LIN {X 0,Y 567.245,Z 796.089,A -85,B 0,C 180,E1 -2627.298,E2 -2627.298} C_VEL
LIN {X 0,Y 567.525,Z 782.898,A -85,B 0,C 180,E1 -2628.314,E2 -2628.314} C_VEL
LIN {X 0,Y 567.877,Z 768.842,A -85,B 0,C 180,E1 -2629.238,E2 -2629.238} C_VEL
LIN {X 0,Y 568.254,Z 752.432,A -85,B 0,C 180,E1 -2630.132,E2 -2630.132} C_VEL
LIN {X 0,Y 568.541,Z 736.853,A -85,B 0,C 180,E1 -2630.817,E2 -2630.817} C_VEL
LIN {X 0,Y 568.789,Z 721.335,A -85,B 0,C 180,E1 -2631.353,E2 -2631.353} C_VEL
LIN {X 0,Y 569.036,Z 705.143,A -85,B 0,C 180,E1 -2631.778,E2 -2631.778} C_VEL
LIN {X 0,Y 569.217,Z 685.553,A -85,B 0,C 180,E1 -2632.108,E2 -2632.108} C_VEL
LIN {X 0,Y 569.98,Z 494.969,A -85,B 0,C 180,E1 -2634.639,E2 -2634.639} C_VEL
LIN {X 0,Y 569.683,Z 492.167,A -85,B 0,C 180,E1 -2634.691,E2 -2634.691} C_VEL
LIN {X 0,Y 567.818,Z 484.792,A -85,B 0,C 180,E1 -2634.886,E2 -2634.886} C_VEL
LIN {X 0,Y 567.716,Z 483.349,A -85,B 0,C 180,E1 -2635.005,E2 -2635.005} C_VEL
LIN {X 0,Y 568.103,Z 461.779,A -85,B 0,C 180,E1 -2637.839,E2 -2637.839} C_VEL
LIN {X 0,Y 568.437,Z 446.604,A -85,B 0,C 180,E1 -2639.873,E2 -2639.873} C_VEL
LIN {X 0,Y 566.233,Z 437.352,A -85,B 0,C 180,E1 -2641.317,E2 -2641.317} C_VEL
LIN {X 0,Y 566.208,Z 437.196,A -85,B 0,C 180,E1 -2643.955,E2 -2643.955} C_VEL
LIN {X 0,Y 566.212,Z 437.2,A -85,B 0,C 180,E1 -2646.568,E2 -2646.568} C_VEL
LIN {X 0,Y 566.207,Z 437.206,A -85,B 0,C 180,E1 -2649.685,E2 -2649.685} C_VEL
LIN {X 0,Y 566.185,Z 437.205,A -85,B 0,C 180,E1 -2652.089,E2 -2652.089} C_VEL
LIN {X 0,Y 566.167,Z 437.206,A -85,B 0,C 180,E1 -2655.035,E2 -2655.035} C_VEL
LIN {X 0,Y 566.208,Z 437.208,A -85,B 0,C 180,E1 -2657.912,E2 -2657.912} C_VEL
LIN {X 0,Y 566.217,Z 437.197,A -85,B 0,C 180,E1 -2660.727,E2 -2660.727} C_VEL
LIN {X 0,Y 566.211,Z 437.207,A -85,B 0,C 180,E1 -2663.783,E2 -2663.783} C_VEL
LIN {X 0,Y 566.204,Z 437.204,A -85,B 0,C 180,E1 -2666.265,E2 -2666.265} C_VEL
LIN {X 0,Y 566.195,Z 437.201,A -85,B 0,C 180,E1 -2668.921,E2 -2668.921} C_VEL
LIN {X 0,Y 566.186,Z 437.196,A -85,B 0,C 180,E1 -2671.046,E2 -2671.046} C_VEL
LIN {X 0,Y 566.236,Z 437.194,A -85,B 0,C 180,E1 -2673.46,E2 -2673.46} C_VEL
LIN {X 0,Y 566.191,Z 437.208,A -85,B 0,C 180,E1 -2675.819,E2 -2675.819} C_VEL
LIN {X 0,Y 566.208,Z 437.192,A -85,B 0,C 180,E1 -2678.902,E2 -2678.902} C_VEL
LIN {X 0,Y 566.204,Z 437.194,A -85,B 0,C 180,E1 -2681.172,E2 -2681.172} C_VEL
LIN {X 0,Y 566.211,Z 437.199,A -85,B 0,C 180,E1 -2683.412,E2 -2683.412} C_VEL
LIN {X 0,Y 566.19,Z 437.208,A -85,B 0,C 180,E1 -2686.359,E2 -2686.359} C_VEL
LIN {X 0,Y 566.266,Z 437.197,A -85,B 0,C 180,E1 -2688.654,E2 -2688.654} C_VEL
LIN {X 0,Y 566.24,Z 437.193,A -85,B 0,C 180,E1 -2691.434,E2 -2691.434} C_VEL
LIN {X 0,Y 566.25,Z 437.203,A -85,B 0,C 180,E1 -2694.302,E2 -2694.302} C_VEL
LIN {X 0,Y 566.271,Z 437.192,A -85,B 0,C 180,E1 -2697.866,E2 -2697.866} C_VEL
LIN {X 0,Y 566.298,Z 437.192,A -85,B 0,C 180,E1 -2700.711,E2 -2700.711} C_VEL
LIN {X 0,Y 566.27,Z 437.197,A -85,B 0,C 180,E1 -2702.845,E2 -2702.845} C_VEL
LIN {X 0,Y 566.258,Z 437.191,A -85,B 0,C 180,E1 -2705.698,E2 -2705.698} C_VEL
LIN {X 0,Y 566.24,Z 437.204,A -85,B 0,C 180,E1 -2708.565,E2 -2708.565} C_VEL
LIN {X 0,Y 566.241,Z 437.194,A -85,B 0,C 180,E1 -2711.454,E2 -2711.454} C_VEL
LIN {X 0,Y 566.223,Z 437.204,A -85,B 0,C 180,E1 -2714.507,E2 -2714.507} C_VEL
LIN {X 0,Y 566.194,Z 437.204,A -85,B 0,C 180,E1 -2717.332,E2 -2717.332} C_VEL
LIN {X 0,Y 566.21,Z 437.201,A -85,B 0,C 180,E1 -2720.337,E2 -2720.337} C_VEL
LIN {X 0,Y 566.18,Z 437.205,A -85,B 0,C 180,E1 -2723.404,E2 -2723.404} C_VEL
LIN {X 0,Y 566.215,Z 437.192,A -85,B 0,C 180,E1 -2725.749,E2 -2725.749} C_VEL
LIN {X 0,Y 566.208,Z 437.198,A -85,B 0,C 180,E1 -2727.495,E2 -2727.495} C_VEL
LIN {X 0,Y 565.53,Z 437.283,A -85,B 0,C 180,E1 -2728.089,E2 -2728.089} C_VEL
LIN {X 0,Y 562.664,Z 437.649,A -85,B 0,C 180,E1 -2729.052,E2 -2729.052} C_VEL
LIN {X 0,Y 560.253,Z 437.945,A -85,B 0,C 180,E1 -2729.828,E2 -2729.828} C_VEL
LIN {X 0,Y 559.224,Z 438.072,A -85,B 0,C 180,E1 -2730.427,E2 -2730.427} C_VEL
LIN {X 0,Y 559.144,Z 438.083,A -85,B 0,C 180,E1 -2730.629,E2 -2730.629} C_VEL
LIN {X 0,Y 559.155,Z 438.071,A -85,B 0,C 180,E1 -2733.575,E2 -2733.575} C_VEL
LIN {X 0,Y 559.16,Z 438.078,A -85,B 0,C 180,E1 -2736.449,E2 -2736.449} C_VEL
LIN {X 0,Y 559.171,Z 438.084,A -85,B 0,C 180,E1 -2738.934,E2 -2738.934} C_VEL
LIN {X 0,Y 559.189,Z 438.077,A -85,B 0,C 180,E1 -2741.767,E2 -2741.767} C_VEL
LIN {X 0,Y 559.132,Z 438.085,A -85,B 0,C 180,E1 -2744.739,E2 -2744.739} C_VEL
LIN {X 0,Y 559.169,Z 438.079,A -85,B 0,C 180,E1 -2747.863,E2 -2747.863} C_VEL
LIN {X 0,Y 559.178,Z 438.076,A -85,B 0,C 180,E1 -2750.135,E2 -2750.135} C_VEL
LIN {X 0,Y 559.14,Z 438.084,A -85,B 0,C 180,E1 -2752.893,E2 -2752.893} C_VEL
LIN {X 0,Y 559.156,Z 438.087,A -85,B 0,C 180,E1 -2755.557,E2 -2755.557} C_VEL
LIN {X 0,Y 559.165,Z 438.079,A -85,B 0,C 180,E1 -2758.138,E2 -2758.138} C_VEL
LIN {X 0,Y 559.138,Z 438.081,A -85,B 0,C 180,E1 -2760.647,E2 -2760.647} C_VEL
LIN {X 0,Y 559.177,Z 438.081,A -85,B 0,C 180,E1 -2763.17,E2 -2763.17} C_VEL
LIN {X 0,Y 559.152,Z 438.088,A -85,B 0,C 180,E1 -2765.495,E2 -2765.495} C_VEL
LIN {X 0,Y 559.167,Z 438.077,A -85,B 0,C 180,E1 -2768.624,E2 -2768.624} C_VEL
LIN {X 0,Y 559.167,Z 438.079,A -85,B 0,C 180,E1 -2770.927,E2 -2770.927} C_VEL
LIN {X 0,Y 559.166,Z 438.085,A -85,B 0,C 180,E1 -2773.948,E2 -2773.948} C_VEL
LIN {X 0,Y 559.171,Z 438.081,A -85,B 0,C 180,E1 -2776.184,E2 -2776.184} C_VEL
LIN {X 0,Y 559.19,Z 438.076,A -85,B 0,C 180,E1 -2779.134,E2 -2779.134} C_VEL
LIN {X 0,Y 559.202,Z 438.081,A -85,B 0,C 180,E1 -2782.054,E2 -2782.054} C_VEL
LIN {X 0,Y 559.249,Z 438.068,A -85,B 0,C 180,E1 -2784.953,E2 -2784.953} C_VEL
LIN {X 0,Y 559.251,Z 438.076,A -85,B 0,C 180,E1 -2787.839,E2 -2787.839} C_VEL
LIN {X 0,Y 559.267,Z 438.066,A -85,B 0,C 180,E1 -2790.72,E2 -2790.72} C_VEL
LIN {X 0,Y 559.235,Z 438.07,A -85,B 0,C 180,E1 -2792.881,E2 -2792.881} C_VEL
LIN {X 0,Y 559.225,Z 438.076,A -85,B 0,C 180,E1 -2795.77,E2 -2795.77} C_VEL
LIN {X 0,Y 559.184,Z 438.078,A -85,B 0,C 180,E1 -2798.674,E2 -2798.674} C_VEL
LIN {X 0,Y 559.202,Z 438.076,A -85,B 0,C 180,E1 -2801.6,E2 -2801.6} C_VEL
LIN {X 0,Y 559.196,Z 438.079,A -85,B 0,C 180,E1 -2804.595,E2 -2804.595} C_VEL
LIN {X 0,Y 559.159,Z 438.079,A -85,B 0,C 180,E1 -2807.556,E2 -2807.556} C_VEL
LIN {X 0,Y 559.168,Z 438.081,A -85,B 0,C 180,E1 -2809.837,E2 -2809.837} C_VEL
LIN {X 0,Y 559.137,Z 438.088,A -85,B 0,C 180,E1 -2812.152,E2 -2812.152} C_VEL
LIN {X 0,Y 559.173,Z 438.077,A -85,B 0,C 180,E1 -2815.298,E2 -2815.298} C_VEL
LIN {X 0,Y 559.19,Z 438.076,A -85,B 0,C 180,E1 -2817.711,E2 -2817.711} C_VEL
LIN {X 0,Y 559.156,Z 438.082,A -85,B 0,C 180,E1 -2821.018,E2 -2821.018} C_VEL
LIN {X 0,Y 559.172,Z 438.079,A -85,B 0,C 180,E1 -2823.951,E2 -2823.951} C_VEL
LIN {X 0,Y 559.162,Z 438.085,A -85,B 0,C 180,E1 -2826.448,E2 -2826.448} C_VEL
LIN {X 0,Y 559.171,Z 438.083,A -85,B 0,C 180,E1 -2828.933,E2 -2828.933} C_VEL
LIN {X 0,Y 559.184,Z 438.075,A -85,B 0,C 180,E1 -2831.767,E2 -2831.767} C_VEL
LIN {X 0,Y 559.132,Z 438.091,A -85,B 0,C 180,E1 -2834.739,E2 -2834.739} C_VEL
LIN {X 0,Y 559.156,Z 438.082,A -85,B 0,C 180,E1 -2837.257,E2 -2837.257} C_VEL
LIN {X 0,Y 559.178,Z 438.077,A -85,B 0,C 180,E1 -2840.135,E2 -2840.135} C_VEL
LIN {X 0,Y 559.139,Z 438.09,A -85,B 0,C 180,E1 -2842.892,E2 -2842.892} C_VEL
LIN {X 0,Y 559.147,Z 438.071,A -85,B 0,C 180,E1 -2845.556,E2 -2845.556} C_VEL
LIN {X 0,Y 559.162,Z 438.076,A -85,B 0,C 180,E1 -2848.137,E2 -2848.137} C_VEL
LIN {X 0,Y 559.149,Z 438.084,A -85,B 0,C 180,E1 -2850.647,E2 -2850.647} C_VEL
LIN {X 0,Y 559.173,Z 438.074,A -85,B 0,C 180,E1 -2853.17,E2 -2853.17} C_VEL
LIN {X 0,Y 559.148,Z 438.082,A -85,B 0,C 180,E1 -2855.495,E2 -2855.495} C_VEL
LIN {X 0,Y 559.167,Z 438.079,A -85,B 0,C 180,E1 -2858.624,E2 -2858.624} C_VEL
LIN {X 0,Y 559.162,Z 438.082,A -85,B 0,C 180,E1 -2860.926,E2 -2860.926} C_VEL
LIN {X 0,Y 559.16,Z 438.075,A -85,B 0,C 180,E1 -2863.948,E2 -2863.948} C_VEL
LIN {X 0,Y 559.163,Z 438.077,A -85,B 0,C 180,E1 -2866.184,E2 -2866.184} C_VEL
LIN {X 0,Y 559.202,Z 438.077,A -85,B 0,C 180,E1 -2869.134,E2 -2869.134} C_VEL
LIN {X 0,Y 559.2,Z 438.073,A -85,B 0,C 180,E1 -2872.054,E2 -2872.054} C_VEL
LIN {X 0,Y 559.253,Z 438.067,A -85,B 0,C 180,E1 -2874.954,E2 -2874.954} C_VEL
LIN {X 0,Y 559.242,Z 438.068,A -85,B 0,C 180,E1 -2877.84,E2 -2877.84} C_VEL
LIN {X 0,Y 559.267,Z 438.065,A -85,B 0,C 180,E1 -2880.72,E2 -2880.72} C_VEL
LIN {X 0,Y 559.236,Z 438.068,A -85,B 0,C 180,E1 -2882.882,E2 -2882.882} C_VEL
LIN {X 0,Y 559.22,Z 438.078,A -85,B 0,C 180,E1 -2885.77,E2 -2885.77} C_VEL
LIN {X 0,Y 559.195,Z 438.07,A -85,B 0,C 180,E1 -2888.674,E2 -2888.674} C_VEL
LIN {X 0,Y 559.2,Z 438.081,A -85,B 0,C 180,E1 -2891.601,E2 -2891.601} C_VEL
LIN {X 0,Y 559.19,Z 438.074,A -85,B 0,C 180,E1 -2894.596,E2 -2894.596} C_VEL
LIN {X 0,Y 559.155,Z 438.084,A -85,B 0,C 180,E1 -2897.557,E2 -2897.557} C_VEL
LIN {X 0,Y 559.166,Z 438.074,A -85,B 0,C 180,E1 -2899.838,E2 -2899.838} C_VEL
LIN {X 0,Y 559.133,Z 438.086,A -85,B 0,C 180,E1 -2902.153,E2 -2902.153} C_VEL
LIN {X 0,Y 559.171,Z 438.077,A -85,B 0,C 180,E1 -2905.188,E2 -2905.188} C_VEL
LIN {X 0,Y 559.186,Z 438.076,A -85,B 0,C 180,E1 -2907.712,E2 -2907.712} C_VEL
LIN {X 0,Y 559.16,Z 438.085,A -85,B 0,C 180,E1 -2910.182,E2 -2910.182} C_VEL
LIN {X 0,Y 559.167,Z 438.078,A -85,B 0,C 180,E1 -2912.714,E2 -2912.714} C_VEL
LIN {X 0,Y 559.149,Z 438.074,A -85,B 0,C 180,E1 -2915.322,E2 -2915.322} C_VEL
LIN {X 0,Y 559.129,Z 438.09,A -85,B 0,C 180,E1 -2918.018,E2 -2918.018} C_VEL
LIN {X 0,Y 559.17,Z 438.078,A -85,B 0,C 180,E1 -2920.811,E2 -2920.811} C_VEL
LIN {X 0,Y 559.156,Z 438.08,A -85,B 0,C 180,E1 -2923.732,E2 -2923.732} C_VEL
LIN {X 0,Y 559.14,Z 438.081,A -85,B 0,C 180,E1 -2926.804,E2 -2926.804} C_VEL
LIN {X 0,Y 559.171,Z 438.078,A -85,B 0,C 180,E1 -2929.19,E2 -2929.19} C_VEL
LIN {X 0,Y 559.129,Z 438.075,A -85,B 0,C 180,E1 -2931.983,E2 -2931.983} C_VEL
LIN {X 0,Y 559.155,Z 438.081,A -85,B 0,C 180,E1 -2934.784,E2 -2934.784} C_VEL
LIN {X 0,Y 559.171,Z 438.078,A -85,B 0,C 180,E1 -2937.362,E2 -2937.362} C_VEL
LIN {X 0,Y 559.189,Z 438.266,A -85,B 0,C 180,E1 -2938.379,E2 -2938.379} C_VEL
LIN {X 0,Y 561.701,Z 448.315,A -85,B 0,C 180,E1 -2939.969,E2 -2939.969} C_VEL
LIN {X 0,Y 561.228,Z 469.907,A -85,B 0,C 180,E1 -2942.89,E2 -2942.89} C_VEL
LIN {X 0,Y 560.941,Z 484.201,A -85,B 0,C 180,E1 -2944.76,E2 -2944.76} C_VEL
LIN {X 0,Y 563.361,Z 494.017,A -85,B 0,C 180,E1 -2945.038,E2 -2945.038} C_VEL
LIN {X 0,Y 563.124,Z 583.687,A -85,B 0,C 180,E1 -2946.257,E2 -2946.257} C_VEL
LIN {X 0,Y 562.553,Z 696.291,A -85,B 0,C 180,E1 -2947.784,E2 -2947.784} C_VEL
LIN {X 0,Y 562.302,Z 712.289,A -85,B 0,C 180,E1 -2948.124,E2 -2948.124} C_VEL
LIN {X 0,Y 562.001,Z 730.611,A -85,B 0,C 180,E1 -2948.689,E2 -2948.689} C_VEL
LIN {X 0,Y 561.681,Z 745.689,A -85,B 0,C 180,E1 -2949.3,E2 -2949.3} C_VEL
LIN {X 0,Y 561.376,Z 758.835,A -85,B 0,C 180,E1 -2949.952,E2 -2949.952} C_VEL
LIN {X 0,Y 560.948,Z 773.325,A -85,B 0,C 180,E1 -2950.8,E2 -2950.8} C_VEL
LIN {X 0,Y 560.595,Z 788.011,A -85,B 0,C 180,E1 -2951.83,E2 -2951.83} C_VEL
LIN {X 0,Y 560.163,Z 802.482,A -85,B 0,C 180,E1 -2953.043,E2 -2953.043} C_VEL
LIN {X 0,Y 559.862,Z 813.823,A -85,B 0,C 180,E1 -2954.156,E2 -2954.156} C_VEL
LIN {X 0,Y 559.584,Z 825.316,A -85,B 0,C 180,E1 -2955.453,E2 -2955.453} C_VEL
LIN {X 0,Y 559.326,Z 836.44,A -85,B 0,C 180,E1 -2956.929,E2 -2956.929} C_VEL
LIN {X 0,Y 559.15,Z 845.808,A -85,B 0,C 180,E1 -2958.399,E2 -2958.399} C_VEL
LIN {X 0,Y 559.013,Z 853.664,A -85,B 0,C 180,E1 -2959.863,E2 -2959.863} C_VEL
LIN {X 0,Y 558.908,Z 860.28,A -85,B 0,C 180,E1 -2961.321,E2 -2961.321} C_VEL
LIN {X 0,Y 558.889,Z 865.667,A -85,B 0,C 180,E1 -2962.776,E2 -2962.776} C_VEL
LIN {X 0,Y 558.863,Z 870.027,A -85,B 0,C 180,E1 -2964.226,E2 -2964.226} C_VEL
LIN {X 0,Y 558.803,Z 873.298,A -85,B 0,C 180,E1 -2965.672,E2 -2965.672} C_VEL
LIN {X 0,Y 558.79,Z 875.656,A -85,B 0,C 180,E1 -2967.116,E2 -2967.116} C_VEL
LIN {X 0,Y 558.738,Z 877.009,A -85,B 0,C 180,E1 -2968.559,E2 -2968.559} C_VEL
LIN {X 0,Y 558.734,Z 877.5,A -85,B 0,C 180,E1 -2970,E2 -2970} C_VEL
LIN {X 0,Y 558.738,Z 877.009,A -85,B 0,C 180,E1 -2971.441,E2 -2971.441} C_VEL
LIN {X 0,Y 558.79,Z 875.656,A -85,B 0,C 180,E1 -2972.884,E2 -2972.884} C_VEL
LIN {X 0,Y 558.802,Z 873.298,A -85,B 0,C 180,E1 -2974.328,E2 -2974.328} C_VEL
LIN {X 0,Y 558.863,Z 870.027,A -85,B 0,C 180,E1 -2975.774,E2 -2975.774} C_VEL
LIN {X 0,Y 558.889,Z 865.667,A -85,B 0,C 180,E1 -2977.224,E2 -2977.224} C_VEL
LIN {X 0,Y 558.908,Z 860.28,A -85,B 0,C 180,E1 -2978.679,E2 -2978.679} C_VEL
LIN {X 0,Y 559.013,Z 853.664,A -85,B 0,C 180,E1 -2980.137,E2 -2980.137} C_VEL
LIN {X 0,Y 559.162,Z 844.729,A -85,B 0,C 180,E1 -2981.785,E2 -2981.785} C_VEL
LIN {X 0,Y 559.359,Z 835.161,A -85,B 0,C 180,E1 -2983.256,E2 -2983.256} C_VEL
LIN {X 0,Y 559.59,Z 825.316,A -85,B 0,C 180,E1 -2984.547,E2 -2984.547} C_VEL
LIN {X 0,Y 559.861,Z 813.823,A -85,B 0,C 180,E1 -2985.844,E2 -2985.844} C_VEL
LIN {X 0,Y 560.199,Z 801.481,A -85,B 0,C 180,E1 -2987.049,E2 -2987.049} C_VEL
LIN {X 0,Y 560.622,Z 786.738,A -85,B 0,C 180,E1 -2988.264,E2 -2988.264} C_VEL
LIN {X 0,Y 560.948,Z 773.325,A -85,B 0,C 180,E1 -2989.2,E2 -2989.2} C_VEL
LIN {X 0,Y 561.341,Z 758.821,A -85,B 0,C 180,E1 -2990.05,E2 -2990.05} C_VEL
LIN {X 0,Y 561.711,Z 743.643,A -85,B 0,C 180,E1 -2990.794,E2 -2990.794} C_VEL
LIN {X 0,Y 562.108,Z 725.885,A -85,B 0,C 180,E1 -2991.475,E2 -2991.475} C_VEL
LIN {X 0,Y 562.367,Z 709.394,A -85,B 0,C 180,E1 -2991.946,E2 -2991.946} C_VEL
LIN {X 0,Y 562.577,Z 693.902,A -85,B 0,C 180,E1 -2992.256,E2 -2992.256} C_VEL
LIN {X 0,Y 563.53,Z 495.969,A -85,B 0,C 180,E1 -2994.927,E2 -2994.927} C_VEL
LIN {X 0,Y 563.082,Z 492.938,A -85,B 0,C 180,E1 -2994.99,E2 -2994.99} C_VEL
LIN {X 0,Y 560.987,Z 484.416,A -85,B 0,C 180,E1 -2995.225,E2 -2995.225} C_VEL
LIN {X 0,Y 561.064,Z 478.235,A -85,B 0,C 180,E1 -2996.002,E2 -2996.002} C_VEL
LIN {X 0,Y 561.525,Z 457.167,A -85,B 0,C 180,E1 -2998.823,E2 -2998.823} C_VEL
LIN {X 0,Y 561.698,Z 448.315,A -85,B 0,C 180,E1 -3000.031,E2 -3000.031} C_VEL
LIN {X 0,Y 559.214,Z 438.272,A -85,B 0,C 180,E1 -3001.619,E2 -3001.619} C_VEL
LIN {X 0,Y 559.153,Z 438.077,A -85,B 0,C 180,E1 -3004.443,E2 -3004.443} C_VEL
LIN {X 0,Y 559.142,Z 438.081,A -85,B 0,C 180,E1 -3007.107,E2 -3007.107} C_VEL
LIN {X 0,Y 559.164,Z 438.085,A -85,B 0,C 180,E1 -3009.942,E2 -3009.942} C_VEL
LIN {X 0,Y 559.152,Z 438.078,A -85,B 0,C 180,E1 -3012.743,E2 -3012.743} C_VEL
LIN {X 0,Y 559.149,Z 438.084,A -85,B 0,C 180,E1 -3015.76,E2 -3015.76} C_VEL
LIN {X 0,Y 559.186,Z 438.077,A -85,B 0,C 180,E1 -3018.232,E2 -3018.232} C_VEL
LIN {X 0,Y 559.172,Z 438.076,A -85,B 0,C 180,E1 -3021.19,E2 -3021.19} C_VEL
LIN {X 0,Y 559.165,Z 438.084,A -85,B 0,C 180,E1 -3023.791,E2 -3023.791} C_VEL
LIN {X 0,Y 559.157,Z 438.08,A -85,B 0,C 180,E1 -3026.425,E2 -3026.425} C_VEL
LIN {X 0,Y 559.158,Z 438.077,A -85,B 0,C 180,E1 -3028.981,E2 -3028.981} C_VEL
LIN {X 0,Y 559.162,Z 438.074,A -85,B 0,C 180,E1 -3031.618,E2 -3031.618} C_VEL
LIN {X 0,Y 559.19,Z 438.077,A -85,B 0,C 180,E1 -3033.903,E2 -3033.903} C_VEL
LIN {X 0,Y 559.148,Z 438.081,A -85,B 0,C 180,E1 -3036.567,E2 -3036.567} C_VEL
LIN {X 0,Y 559.177,Z 438.067,A -85,B 0,C 180,E1 -3039.395,E2 -3039.395} C_VEL
LIN {X 0,Y 559.146,Z 438.075,A -85,B 0,C 180,E1 -3041.686,E2 -3041.686} C_VEL
LIN {X 0,Y 559.161,Z 438.082,A -85,B 0,C 180,E1 -3043.948,E2 -3043.948} C_VEL
LIN {X 0,Y 559.164,Z 438.084,A -85,B 0,C 180,E1 -3046.184,E2 -3046.184} C_VEL
LIN {X 0,Y 559.202,Z 438.073,A -85,B 0,C 180,E1 -3049.134,E2 -3049.134} C_VEL
LIN {X 0,Y 559.2,Z 438.074,A -85,B 0,C 180,E1 -3052.053,E2 -3052.053} C_VEL
LIN {X 0,Y 559.251,Z 438.067,A -85,B 0,C 180,E1 -3054.953,E2 -3054.953} C_VEL
LIN {X 0,Y 559.243,Z 438.068,A -85,B 0,C 180,E1 -3057.839,E2 -3057.839} C_VEL
LIN {X 0,Y 559.267,Z 438.067,A -85,B 0,C 180,E1 -3060.72,E2 -3060.72} C_VEL
LIN {X 0,Y 559.236,Z 438.072,A -85,B 0,C 180,E1 -3062.881,E2 -3062.881} C_VEL
LIN {X 0,Y 559.227,Z 438.067,A -85,B 0,C 180,E1 -3065.77,E2 -3065.77} C_VEL
LIN {X 0,Y 559.195,Z 438.082,A -85,B 0,C 180,E1 -3068.674,E2 -3068.674} C_VEL
LIN {X 0,Y 559.199,Z 438.07,A -85,B 0,C 180,E1 -3071.6,E2 -3071.6} C_VEL
LIN {X 0,Y 559.189,Z 438.082,A -85,B 0,C 180,E1 -3074.596,E2 -3074.596} C_VEL
LIN {X 0,Y 559.154,Z 438.079,A -85,B 0,C 180,E1 -3077.557,E2 -3077.557} C_VEL
LIN {X 0,Y 559.165,Z 438.076,A -85,B 0,C 180,E1 -3079.837,E2 -3079.837} C_VEL
LIN {X 0,Y 559.132,Z 438.082,A -85,B 0,C 180,E1 -3082.153,E2 -3082.153} C_VEL
LIN {X 0,Y 559.17,Z 438.074,A -85,B 0,C 180,E1 -3085.187,E2 -3085.187} C_VEL
LIN {X 0,Y 559.186,Z 438.07,A -85,B 0,C 180,E1 -3087.712,E2 -3087.712} C_VEL
LIN {X 0,Y 559.144,Z 438.083,A -85,B 0,C 180,E1 -3090.629,E2 -3090.629} C_VEL
LIN {X 0,Y 558.481,Z 438.171,A -85,B 0,C 180,E1 -3091.231,E2 -3091.231} C_VEL
LIN {X 0,Y 555.615,Z 438.523,A -85,B 0,C 180,E1 -3092.207,E2 -3092.207} C_VEL
LIN {X 0,Y 553.201,Z 438.821,A -85,B 0,C 180,E1 -3092.993,E2 -3092.993} C_VEL
LIN {X 0,Y 552.18,Z 438.939,A -85,B 0,C 180,E1 -3093.599,E2 -3093.599} C_VEL
LIN {X 0,Y 552.106,Z 438.946,A -85,B 0,C 180,E1 -3093.805,E2 -3093.805} C_VEL
LIN {X 0,Y 552.103,Z 438.96,A -85,B 0,C 180,E1 -3096.747,E2 -3096.747} C_VEL
LIN {X 0,Y 552.127,Z 438.959,A -85,B 0,C 180,E1 -3099.527,E2 -3099.527} C_VEL
LIN {X 0,Y 552.162,Z 438.956,A -85,B 0,C 180,E1 -3101.442,E2 -3101.442} C_VEL
LIN {X 0,Y 552.088,Z 438.96,A -85,B 0,C 180,E1 -3104.532,E2 -3104.532} C_VEL
LIN {X 0,Y 552.123,Z 438.96,A -85,B 0,C 180,E1 -3107.585,E2 -3107.585} C_VEL
LIN {X 0,Y 552.127,Z 438.955,A -85,B 0,C 180,E1 -3110.474,E2 -3110.474} C_VEL
LIN {X 0,Y 552.108,Z 438.965,A -85,B 0,C 180,E1 -3113.316,E2 -3113.316} C_VEL
LIN {X 0,Y 552.134,Z 438.957,A -85,B 0,C 180,E1 -3115.941,E2 -3115.941} C_VEL
LIN {X 0,Y 552.113,Z 438.957,A -85,B 0,C 180,E1 -3118.541,E2 -3118.541} C_VEL
LIN {X 0,Y 552.121,Z 438.964,A -85,B 0,C 180,E1 -3121.438,E2 -3121.438} C_VEL
LIN {X 0,Y 552.132,Z 438.954,A -85,B 0,C 180,E1 -3124.357,E2 -3124.357} C_VEL
LIN {X 0,Y 552.105,Z 438.958,A -85,B 0,C 180,E1 -3126.759,E2 -3126.759} C_VEL
LIN {X 0,Y 552.116,Z 438.958,A -85,B 0,C 180,E1 -3129.12,E2 -3129.12} C_VEL
LIN {X 0,Y 552.127,Z 438.962,A -85,B 0,C 180,E1 -3131.445,E2 -3131.445} C_VEL
LIN {X 0,Y 552.116,Z 438.965,A -85,B 0,C 180,E1 -3133.738,E2 -3133.738} C_VEL
LIN {X 0,Y 552.133,Z 438.96,A -85,B 0,C 180,E1 -3136.005,E2 -3136.005} C_VEL
LIN {X 0,Y 552.158,Z 438.952,A -85,B 0,C 180,E1 -3138.994,E2 -3138.994} C_VEL
LIN {X 0,Y 552.156,Z 438.959,A -85,B 0,C 180,E1 -3141.952,E2 -3141.952} C_VEL
LIN {X 0,Y 552.224,Z 438.943,A -85,B 0,C 180,E1 -3144.889,E2 -3144.889} C_VEL
LIN {X 0,Y 552.222,Z 438.951,A -85,B 0,C 180,E1 -3147.812,E2 -3147.812} C_VEL
LIN {X 0,Y 552.238,Z 438.942,A -85,B 0,C 180,E1 -3150.729,E2 -3150.729} C_VEL
LIN {X 0,Y 552.202,Z 438.946,A -85,B 0,C 180,E1 -3152.918,E2 -3152.918} C_VEL
LIN {X 0,Y 552.195,Z 438.953,A -85,B 0,C 180,E1 -3155.844,E2 -3155.844} C_VEL
LIN {X 0,Y 552.155,Z 438.953,A -85,B 0,C 180,E1 -3158.786,E2 -3158.786} C_VEL
LIN {X 0,Y 552.159,Z 438.955,A -85,B 0,C 180,E1 -3161.75,E2 -3161.75} C_VEL
LIN {X 0,Y 552.133,Z 438.957,A -85,B 0,C 180,E1 -3164.748,E2 -3164.748} C_VEL
LIN {X 0,Y 552.111,Z 438.959,A -85,B 0,C 180,E1 -3167.788,E2 -3167.788} C_VEL
LIN {X 0,Y 552.127,Z 438.962,A -85,B 0,C 180,E1 -3170.101,E2 -3170.101} C_VEL
LIN {X 0,Y 552.088,Z 438.968,A -85,B 0,C 180,E1 -3172.451,E2 -3172.451} C_VEL
LIN {X 0,Y 552.152,Z 438.952,A -85,B 0,C 180,E1 -3175.35,E2 -3175.35} C_VEL
LIN {X 0,Y 552.122,Z 438.96,A -85,B 0,C 180,E1 -3178.097,E2 -3178.097} C_VEL
LIN {X 0,Y 552.101,Z 438.966,A -85,B 0,C 180,E1 -3180.609,E2 -3180.609} C_VEL
LIN {X 0,Y 552.123,Z 438.957,A -85,B 0,C 180,E1 -3183.184,E2 -3183.184} C_VEL
LIN {X 0,Y 552.107,Z 438.957,A -85,B 0,C 180,E1 -3185.841,E2 -3185.841} C_VEL
LIN {X 0,Y 552.118,Z 438.96,A -85,B 0,C 180,E1 -3189.061,E2 -3189.061} C_VEL
LIN {X 0,Y 552.132,Z 438.955,A -85,B 0,C 180,E1 -3191.444,E2 -3191.444} C_VEL
LIN {X 0,Y 552.088,Z 438.966,A -85,B 0,C 180,E1 -3194.532,E2 -3194.532} C_VEL
LIN {X 0,Y 552.123,Z 438.956,A -85,B 0,C 180,E1 -3197.584,E2 -3197.584} C_VEL
LIN {X 0,Y 552.135,Z 438.954,A -85,B 0,C 180,E1 -3199.792,E2 -3199.792} C_VEL
LIN {X 0,Y 552.086,Z 438.962,A -85,B 0,C 180,E1 -3202.336,E2 -3202.336} C_VEL
LIN {X 0,Y 552.12,Z 438.952,A -85,B 0,C 180,E1 -3205.054,E2 -3205.054} C_VEL
LIN {X 0,Y 552.118,Z 438.954,A -85,B 0,C 180,E1 -3207.682,E2 -3207.682} C_VEL
LIN {X 0,Y 552.136,Z 438.954,A -85,B 0,C 180,E1 -3210.237,E2 -3210.237} C_VEL
LIN {X 0,Y 552.138,Z 438.949,A -85,B 0,C 180,E1 -3212.998,E2 -3212.998} C_VEL
LIN {X 0,Y 552.104,Z 438.96,A -85,B 0,C 180,E1 -3215.161,E2 -3215.161} C_VEL
LIN {X 0,Y 552.086,Z 438.963,A -85,B 0,C 180,E1 -3217.549,E2 -3217.549} C_VEL
LIN {X 0,Y 552.139,Z 438.951,A -85,B 0,C 180,E1 -3220.373,E2 -3220.373} C_VEL
LIN {X 0,Y 552.147,Z 438.958,A -85,B 0,C 180,E1 -3222.977,E2 -3222.977} C_VEL
LIN {X 0,Y 552.126,Z 438.954,A -85,B 0,C 180,E1 -3226.004,E2 -3226.004} C_VEL
LIN {X 0,Y 552.169,Z 438.95,A -85,B 0,C 180,E1 -3228.994,E2 -3228.994} C_VEL
LIN {X 0,Y 552.154,Z 438.951,A -85,B 0,C 180,E1 -3231.952,E2 -3231.952} C_VEL
LIN {X 0,Y 552.227,Z 438.941,A -85,B 0,C 180,E1 -3234.889,E2 -3234.889} C_VEL
LIN {X 0,Y 552.214,Z 438.944,A -85,B 0,C 180,E1 -3237.812,E2 -3237.812} C_VEL
LIN {X 0,Y 552.237,Z 438.941,A -85,B 0,C 180,E1 -3240.729,E2 -3240.729} C_VEL
LIN {X 0,Y 552.202,Z 438.945,A -85,B 0,C 180,E1 -3242.918,E2 -3242.918} C_VEL
LIN {X 0,Y 552.19,Z 438.952,A -85,B 0,C 180,E1 -3245.844,E2 -3245.844} C_VEL
LIN {X 0,Y 552.162,Z 438.945,A -85,B 0,C 180,E1 -3248.786,E2 -3248.786} C_VEL
LIN {X 0,Y 552.155,Z 438.958,A -85,B 0,C 180,E1 -3251.751,E2 -3251.751} C_VEL
LIN {X 0,Y 552.127,Z 438.953,A -85,B 0,C 180,E1 -3254.749,E2 -3254.749} C_VEL
LIN {X 0,Y 552.106,Z 438.96,A -85,B 0,C 180,E1 -3257.789,E2 -3257.789} C_VEL
LIN {X 0,Y 552.125,Z 438.948,A -85,B 0,C 180,E1 -3260.101,E2 -3260.101} C_VEL
LIN {X 0,Y 552.087,Z 438.959,A -85,B 0,C 180,E1 -3262.451,E2 -3262.451} C_VEL
LIN {X 0,Y 552.148,Z 438.953,A -85,B 0,C 180,E1 -3265.351,E2 -3265.351} C_VEL
LIN {X 0,Y 552.118,Z 438.951,A -85,B 0,C 180,E1 -3268.098,E2 -3268.098} C_VEL
LIN {X 0,Y 552.106,Z 438.958,A -85,B 0,C 180,E1 -3270.609,E2 -3270.609} C_VEL
LIN {X 0,Y 552.115,Z 438.955,A -85,B 0,C 180,E1 -3273.186,E2 -3273.186} C_VEL
LIN {X 0,Y 552.105,Z 438.956,A -85,B 0,C 180,E1 -3275.842,E2 -3275.842} C_VEL
LIN {X 0,Y 552.12,Z 438.953,A -85,B 0,C 180,E1 -3279.063,E2 -3279.063} C_VEL
LIN {X 0,Y 552.134,Z 438.953,A -85,B 0,C 180,E1 -3281.445,E2 -3281.445} C_VEL
LIN {X 0,Y 552.09,Z 438.964,A -85,B 0,C 180,E1 -3284.533,E2 -3284.533} C_VEL
LIN {X 0,Y 552.125,Z 438.953,A -85,B 0,C 180,E1 -3287.585,E2 -3287.585} C_VEL
LIN {X 0,Y 552.129,Z 438.954,A -85,B 0,C 180,E1 -3290.474,E2 -3290.474} C_VEL
LIN {X 0,Y 552.11,Z 438.957,A -85,B 0,C 180,E1 -3293.316,E2 -3293.316} C_VEL
LIN {X 0,Y 552.128,Z 438.946,A -85,B 0,C 180,E1 -3295.94,E2 -3295.94} C_VEL
LIN {X 0,Y 552.157,Z 439.176,A -85,B 0,C 180,E1 -3298.062,E2 -3298.062} C_VEL
LIN {X 0,Y 554.802,Z 449.38,A -85,B 0,C 180,E1 -3299.706,E2 -3299.706} C_VEL
LIN {X 0,Y 554.917,Z 454.299,A -85,B 0,C 180,E1 -3300.401,E2 -3300.401} C_VEL
LIN {X 0,Y 554.342,Z 475.243,A -85,B 0,C 180,E1 -3303.252,E2 -3303.252} C_VEL
LIN {X 0,Y 554.176,Z 484.209,A -85,B 0,C 180,E1 -3304.431,E2 -3304.431} C_VEL
LIN {X 0,Y 556.799,Z 494.797,A -85,B 0,C 180,E1 -3304.735,E2 -3304.735} C_VEL
LIN {X 0,Y 557.085,Z 498.55,A -85,B 0,C 180,E1 -3304.801,E2 -3304.801} C_VEL
LIN {X 0,Y 556.079,Z 686.065,A -85,B 0,C 180,E1 -3307.348,E2 -3307.348} C_VEL
LIN {X 0,Y 555.859,Z 704.784,A -85,B 0,C 180,E1 -3307.671,E2 -3307.671} C_VEL
LIN {X 0,Y 555.574,Z 720.547,A -85,B 0,C 180,E1 -3308.089,E2 -3308.089} C_VEL
LIN {X 0,Y 555.246,Z 735.59,A -85,B 0,C 180,E1 -3308.612,E2 -3308.612} C_VEL
LIN {X 0,Y 554.873,Z 749.759,A -85,B 0,C 180,E1 -3309.229,E2 -3309.229} C_VEL
LIN {X 0,Y 554.415,Z 767.286,A -85,B 0,C 180,E1 -3310.179,E2 -3310.179} C_VEL
LIN {X 0,Y 554.002,Z 780.284,A -85,B 0,C 180,E1 -3311.03,E2 -3311.03} C_VEL
LIN {X 0,Y 553.62,Z 792.665,A -85,B 0,C 180,E1 -3311.976,E2 -3311.976} C_VEL
LIN {X 0,Y 553.187,Z 804.447,A -85,B 0,C 180,E1 -3313.01,E2 -3313.01} C_VEL
LIN {X 0,Y 552.894,Z 815.582,A -85,B 0,C 180,E1 -3314.14,E2 -3314.14} C_VEL
LIN {X 0,Y 552.589,Z 826.809,A -85,B 0,C 180,E1 -3315.453,E2 -3315.453} C_VEL
LIN {X 0,Y 552.301,Z 837.68,A -85,B 0,C 180,E1 -3316.946,E2 -3316.946} C_VEL
LIN {X 0,Y 552.112,Z 845.803,A -85,B 0,C 180,E1 -3318.249,E2 -3318.249} C_VEL
LIN {X 0,Y 551.956,Z 853.661,A -85,B 0,C 180,E1 -3319.732,E2 -3319.732} C_VEL
LIN {X 0,Y 551.834,Z 860.275,A -85,B 0,C 180,E1 -3321.209,E2 -3321.209} C_VEL
LIN {X 0,Y 551.807,Z 865.667,A -85,B 0,C 180,E1 -3322.683,E2 -3322.683} C_VEL
LIN {X 0,Y 551.77,Z 870.026,A -85,B 0,C 180,E1 -3324.152,E2 -3324.152} C_VEL
LIN {X 0,Y 551.699,Z 873.3,A -85,B 0,C 180,E1 -3325.617,E2 -3325.617} C_VEL
LIN {X 0,Y 551.714,Z 875.656,A -85,B 0,C 180,E1 -3327.079,E2 -3327.079} C_VEL
LIN {X 0,Y 551.638,Z 877.011,A -85,B 0,C 180,E1 -3328.54,E2 -3328.54} C_VEL
LIN {X 0,Y 551.635,Z 877.5,A -85,B 0,C 180,E1 -3330,E2 -3330} C_VEL
LIN {X 0,Y 551.638,Z 877.011,A -85,B 0,C 180,E1 -3331.46,E2 -3331.46} C_VEL
LIN {X 0,Y 551.714,Z 875.656,A -85,B 0,C 180,E1 -3332.921,E2 -3332.921} C_VEL
LIN {X 0,Y 551.698,Z 873.3,A -85,B 0,C 180,E1 -3334.383,E2 -3334.383} C_VEL
LIN {X 0,Y 551.77,Z 870.026,A -85,B 0,C 180,E1 -3335.848,E2 -3335.848} C_VEL
LIN {X 0,Y 551.807,Z 865.667,A -85,B 0,C 180,E1 -3337.317,E2 -3337.317} C_VEL
LIN {X 0,Y 551.834,Z 860.275,A -85,B 0,C 180,E1 -3338.791,E2 -3338.791} C_VEL
LIN {X 0,Y 551.956,Z 853.661,A -85,B 0,C 180,E1 -3340.268,E2 -3340.268} C_VEL
LIN {X 0,Y 552.103,Z 845.803,A -85,B 0,C 180,E1 -3341.751,E2 -3341.751} C_VEL
LIN {X 0,Y 552.358,Z 835.159,A -85,B 0,C 180,E1 -3343.427,E2 -3343.427} C_VEL
LIN {X 0,Y 552.668,Z 824.077,A -85,B 0,C 180,E1 -3344.884,E2 -3344.884} C_VEL
LIN {X 0,Y 552.93,Z 813.818,A -85,B 0,C 180,E1 -3346.048,E2 -3346.048} C_VEL
LIN {X 0,Y 553.341,Z 800.812,A -85,B 0,C 180,E1 -3347.329,E2 -3347.329} C_VEL
LIN {X 0,Y 553.791,Z 786.738,A -85,B 0,C 180,E1 -3348.497,E2 -3348.497} C_VEL
LIN {X 0,Y 554.193,Z 773.314,A -85,B 0,C 180,E1 -3349.444,E2 -3349.444} C_VEL
LIN {X 0,Y 554.59,Z 759.605,A -85,B 0,C 180,E1 -3350.261,E2 -3350.261} C_VEL
LIN {X 0,Y 554.997,Z 745.676,A -85,B 0,C 180,E1 -3350.961,E2 -3350.961} C_VEL
LIN {X 0,Y 555.387,Z 730.616,A -85,B 0,C 180,E1 -3351.577,E2 -3351.577} C_VEL
LIN {X 0,Y 555.751,Z 712.299,A -85,B 0,C 180,E1 -3352.148,E2 -3352.148} C_VEL
LIN {X 0,Y 555.982,Z 696.099,A -85,B 0,C 180,E1 -3352.496,E2 -3352.496} C_VEL
LIN {X 0,Y 557.011,Z 513.856,A -85,B 0,C 180,E1 -3354.989,E2 -3354.989} C_VEL
LIN {X 0,Y 557.042,Z 495.777,A -85,B 0,C 180,E1 -3355.24,E2 -3355.24} C_VEL
LIN {X 0,Y 554.215,Z 484.406,A -85,B 0,C 180,E1 -3355.554,E2 -3355.554} C_VEL
LIN {X 0,Y 554.485,Z 470.827,A -85,B 0,C 180,E1 -3357.342,E2 -3357.342} C_VEL
LIN {X 0,Y 554.977,Z 451.307,A -85,B 0,C 180,E1 -3360.013,E2 -3360.013} C_VEL
LIN {X 0,Y 554.15,Z 446.822,A -85,B 0,C 180,E1 -3360.694,E2 -3360.694} C_VEL
LIN {X 0,Y 552.138,Z 439.085,A -85,B 0,C 180,E1 -3361.966,E2 -3361.966} C_VEL
LIN {X 0,Y 552.125,Z 438.953,A -85,B 0,C 180,E1 -3364.945,E2 -3364.945} C_VEL
LIN {X 0,Y 552.092,Z 438.95,A -85,B 0,C 180,E1 -3367.885,E2 -3367.885} C_VEL
LIN {X 0,Y 552.116,Z 438.958,A -85,B 0,C 180,E1 -3370.479,E2 -3370.479} C_VEL
LIN {X 0,Y 552.096,Z 438.963,A -85,B 0,C 180,E1 -3373.482,E2 -3373.482} C_VEL
LIN {X 0,Y 552.114,Z 438.955,A -85,B 0,C 180,E1 -3376.577,E2 -3376.577} C_VEL
LIN {X 0,Y 552.136,Z 438.958,A -85,B 0,C 180,E1 -3379.521,E2 -3379.521} C_VEL
LIN {X 0,Y 552.088,Z 438.962,A -85,B 0,C 180,E1 -3382.336,E2 -3382.336} C_VEL
LIN {X 0,Y 552.121,Z 438.948,A -85,B 0,C 180,E1 -3385.054,E2 -3385.054} C_VEL
LIN {X 0,Y 552.12,Z 438.96,A -85,B 0,C 180,E1 -3387.682,E2 -3387.682} C_VEL
LIN {X 0,Y 552.137,Z 438.95,A -85,B 0,C 180,E1 -3390.237,E2 -3390.237} C_VEL
LIN {X 0,Y 552.139,Z 438.947,A -85,B 0,C 180,E1 -3392.998,E2 -3392.998} C_VEL
LIN {X 0,Y 552.105,Z 438.957,A -85,B 0,C 180,E1 -3395.161,E2 -3395.161} C_VEL
LIN {X 0,Y 552.087,Z 438.959,A -85,B 0,C 180,E1 -3397.549,E2 -3397.549} C_VEL
LIN {X 0,Y 552.14,Z 438.948,A -85,B 0,C 180,E1 -3400.373,E2 -3400.373} C_VEL
LIN {X 0,Y 552.148,Z 438.951,A -85,B 0,C 180,E1 -3402.977,E2 -3402.977} C_VEL
LIN {X 0,Y 552.127,Z 438.959,A -85,B 0,C 180,E1 -3406.004,E2 -3406.004} C_VEL
LIN {X 0,Y 552.169,Z 438.949,A -85,B 0,C 180,E1 -3408.993,E2 -3408.993} C_VEL
LIN {X 0,Y 552.154,Z 438.95,A -85,B 0,C 180,E1 -3411.951,E2 -3411.951} C_VEL
LIN {X 0,Y 552.225,Z 438.943,A -85,B 0,C 180,E1 -3414.889,E2 -3414.889} C_VEL
LIN {X 0,Y 552.214,Z 438.943,A -85,B 0,C 180,E1 -3417.812,E2 -3417.812} C_VEL
LIN {X 0,Y 552.237,Z 438.942,A -85,B 0,C 180,E1 -3420.729,E2 -3420.729} C_VEL
LIN {X 0,Y 552.202,Z 438.948,A -85,B 0,C 180,E1 -3422.918,E2 -3422.918} C_VEL
LIN {X 0,Y 552.197,Z 438.943,A -85,B 0,C 180,E1 -3425.844,E2 -3425.844} C_VEL
LIN {X 0,Y 552.162,Z 438.956,A -85,B 0,C 180,E1 -3428.785,E2 -3428.785} C_VEL
LIN {X 0,Y 552.155,Z 438.947,A -85,B 0,C 180,E1 -3431.75,E2 -3431.75} C_VEL
LIN {X 0,Y 552.126,Z 438.961,A -85,B 0,C 180,E1 -3434.748,E2 -3434.748} C_VEL
LIN {X 0,Y 552.105,Z 438.957,A -85,B 0,C 180,E1 -3437.788,E2 -3437.788} C_VEL
LIN {X 0,Y 552.124,Z 438.953,A -85,B 0,C 180,E1 -3440.101,E2 -3440.101} C_VEL
LIN {X 0,Y 552.086,Z 438.963,A -85,B 0,C 180,E1 -3442.451,E2 -3442.451} C_VEL
LIN {X 0,Y 552.147,Z 438.946,A -85,B 0,C 180,E1 -3445.351,E2 -3445.351} C_VEL
LIN {X 0,Y 552.117,Z 438.95,A -85,B 0,C 180,E1 -3448.098,E2 -3448.098} C_VEL
LIN {X 0,Y 552.104,Z 438.961,A -85,B 0,C 180,E1 -3450.625,E2 -3450.625} C_VEL
LIN {X 0,Y 552.113,Z 438.952,A -85,B 0,C 180,E1 -3453.186,E2 -3453.186} C_VEL
LIN {X 0,Y 552.106,Z 438.946,A -85,B 0,C 180,E1 -3453.805,E2 -3453.805} C_VEL
LIN {X 0,Y 551.464,Z 439.028,A -85,B 0,C 180,E1 -3454.413,E2 -3454.413} C_VEL
LIN {X 0,Y 548.62,Z 439.395,A -85,B 0,C 180,E1 -3455.401,E2 -3455.401} C_VEL
LIN {X 0,Y 546.198,Z 439.699,A -85,B 0,C 180,E1 -3456.197,E2 -3456.197} C_VEL
LIN {X 0,Y 545.151,Z 439.829,A -85,B 0,C 180,E1 -3456.811,E2 -3456.811} C_VEL
LIN {X 0,Y 545.063,Z 439.84,A -85,B 0,C 180,E1 -3457.019,E2 -3457.019} C_VEL
LIN {X 0,Y 545.086,Z 439.832,A -85,B 0,C 180,E1 -3460.14,E2 -3460.14} C_VEL
LIN {X 0,Y 545.058,Z 439.838,A -85,B 0,C 180,E1 -3462.698,E2 -3462.698} C_VEL
LIN {X 0,Y 545.055,Z 439.844,A -85,B 0,C 180,E1 -3465.167,E2 -3465.167} C_VEL
LIN {X 0,Y 545.075,Z 439.835,A -85,B 0,C 180,E1 -3467.898,E2 -3467.898} C_VEL
LIN {X 0,Y 545.098,Z 439.832,A -85,B 0,C 180,E1 -3470.676,E2 -3470.676} C_VEL
LIN {X 0,Y 545.049,Z 439.842,A -85,B 0,C 180,E1 -3473.621,E2 -3473.621} C_VEL
LIN {X 0,Y 545.072,Z 439.834,A -85,B 0,C 180,E1 -3476.329,E2 -3476.329} C_VEL
LIN {X 0,Y 545.062,Z 439.837,A -85,B 0,C 180,E1 -3478.953,E2 -3478.953} C_VEL
LIN {X 0,Y 545.099,Z 439.838,A -85,B 0,C 180,E1 -3481.508,E2 -3481.508} C_VEL
LIN {X 0,Y 545.094,Z 439.831,A -85,B 0,C 180,E1 -3484.49,E2 -3484.49} C_VEL
LIN {X 0,Y 545.04,Z 439.842,A -85,B 0,C 180,E1 -3487.243,E2 -3487.243} C_VEL
LIN {X 0,Y 545.116,Z 439.83,A -85,B 0,C 180,E1 -3490.415,E2 -3490.415} C_VEL
LIN {X 0,Y 545.072,Z 439.84,A -85,B 0,C 180,E1 -3493.522,E2 -3493.522} C_VEL
LIN {X 0,Y 545.092,Z 439.84,A -85,B 0,C 180,E1 -3495.82,E2 -3495.82} C_VEL
LIN {X 0,Y 545.114,Z 439.829,A -85,B 0,C 180,E1 -3498.85,E2 -3498.85} C_VEL
LIN {X 0,Y 545.126,Z 439.836,A -85,B 0,C 180,E1 -3501.847,E2 -3501.847} C_VEL
LIN {X 0,Y 545.2,Z 439.818,A -85,B 0,C 180,E1 -3504.823,E2 -3504.823} C_VEL
LIN {X 0,Y 545.194,Z 439.827,A -85,B 0,C 180,E1 -3507.784,E2 -3507.784} C_VEL
LIN {X 0,Y 545.208,Z 439.818,A -85,B 0,C 180,E1 -3510.739,E2 -3510.739} C_VEL
LIN {X 0,Y 545.169,Z 439.823,A -85,B 0,C 180,E1 -3512.956,E2 -3512.956} C_VEL
LIN {X 0,Y 545.167,Z 439.83,A -85,B 0,C 180,E1 -3515.919,E2 -3515.919} C_VEL
LIN {X 0,Y 545.114,Z 439.829,A -85,B 0,C 180,E1 -3518.9,E2 -3518.9} C_VEL
LIN {X 0,Y 545.132,Z 439.832,A -85,B 0,C 180,E1 -3521.904,E2 -3521.904} C_VEL
LIN {X 0,Y 545.082,Z 439.834,A -85,B 0,C 180,E1 -3524.943,E2 -3524.943} C_VEL
LIN {X 0,Y 545.079,Z 439.838,A -85,B 0,C 180,E1 -3528.025,E2 -3528.025} C_VEL
LIN {X 0,Y 545.091,Z 439.84,A -85,B 0,C 180,E1 -3530.372,E2 -3530.372} C_VEL
LIN {X 0,Y 545.076,Z 439.834,A -85,B 0,C 180,E1 -3533.559,E2 -3533.559} C_VEL
LIN {X 0,Y 545.084,Z 439.836,A -85,B 0,C 180,E1 -3536,E2 -3536} C_VEL
LIN {X 0,Y 545.085,Z 439.838,A -85,B 0,C 180,E1 -3538.748,E2 -3538.748} C_VEL
LIN {X 0,Y 545.072,Z 439.834,A -85,B 0,C 180,E1 -3541.682,E2 -3541.682} C_VEL
LIN {X 0,Y 545.079,Z 439.841,A -85,B 0,C 180,E1 -3544.562,E2 -3544.562} C_VEL
LIN {X 0,Y 545.032,Z 439.84,A -85,B 0,C 180,E1 -3547.303,E2 -3547.303} C_VEL
LIN {X 0,Y 545.085,Z 439.834,A -85,B 0,C 180,E1 -3550.14,E2 -3550.14} C_VEL
LIN {X 0,Y 545.07,Z 439.838,A -85,B 0,C 180,E1 -3553.106,E2 -3553.106} C_VEL
LIN {X 0,Y 545.056,Z 439.838,A -85,B 0,C 180,E1 -3556.224,E2 -3556.224} C_VEL
LIN {X 0,Y 545.114,Z 439.837,A -85,B 0,C 180,E1 -3558.889,E2 -3558.889} C_VEL
LIN {X 0,Y 545.046,Z 439.837,A -85,B 0,C 180,E1 -3561.763,E2 -3561.763} C_VEL
LIN {X 0,Y 545.056,Z 439.838,A -85,B 0,C 180,E1 -3564.534,E2 -3564.534} C_VEL
LIN {X 0,Y 545.072,Z 439.837,A -85,B 0,C 180,E1 -3567.212,E2 -3567.212} C_VEL
LIN {X 0,Y 545.092,Z 439.831,A -85,B 0,C 180,E1 -3569.813,E2 -3569.813} C_VEL
LIN {X 0,Y 545.092,Z 439.827,A -85,B 0,C 180,E1 -3572.824,E2 -3572.824} C_VEL
LIN {X 0,Y 545.043,Z 439.838,A -85,B 0,C 180,E1 -3575.631,E2 -3575.631} C_VEL
LIN {X 0,Y 545.06,Z 439.839,A -85,B 0,C 180,E1 -3578.837,E2 -3578.837} C_VEL
LIN {X 0,Y 545.076,Z 439.841,A -85,B 0,C 180,E1 -3581.196,E2 -3581.196} C_VEL
LIN {X 0,Y 545.066,Z 439.835,A -85,B 0,C 180,E1 -3583.521,E2 -3583.521} C_VEL
LIN {X 0,Y 545.085,Z 439.833,A -85,B 0,C 180,E1 -3585.82,E2 -3585.82} C_VEL
LIN {X 0,Y 545.123,Z 439.826,A -85,B 0,C 180,E1 -3588.85,E2 -3588.85} C_VEL
LIN {X 0,Y 545.124,Z 439.828,A -85,B 0,C 180,E1 -3591.847,E2 -3591.847} C_VEL
LIN {X 0,Y 545.202,Z 439.816,A -85,B 0,C 180,E1 -3594.823,E2 -3594.823} C_VEL
LIN {X 0,Y 545.186,Z 439.819,A -85,B 0,C 180,E1 -3597.784,E2 -3597.784} C_VEL
LIN {X 0,Y 545.207,Z 439.817,A -85,B 0,C 180,E1 -3600.739,E2 -3600.739} C_VEL
LIN {X 0,Y 545.168,Z 439.821,A -85,B 0,C 180,E1 -3602.956,E2 -3602.956} C_VEL
LIN {X 0,Y 545.162,Z 439.826,A -85,B 0,C 180,E1 -3605.92,E2 -3605.92} C_VEL
LIN {X 0,Y 545.119,Z 439.823,A -85,B 0,C 180,E1 -3608.9,E2 -3608.9} C_VEL
LIN {X 0,Y 545.127,Z 439.83,A -85,B 0,C 180,E1 -3611.904,E2 -3611.904} C_VEL
LIN {X 0,Y 545.076,Z 439.832,A -85,B 0,C 180,E1 -3614.944,E2 -3614.944} C_VEL
LIN {X 0,Y 545.074,Z 439.83,A -85,B 0,C 180,E1 -3618.026,E2 -3618.026} C_VEL
LIN {X 0,Y 545.09,Z 439.822,A -85,B 0,C 180,E1 -3620.372,E2 -3620.372} C_VEL
LIN {X 0,Y 545.083,Z 439.834,A -85,B 0,C 180,E1 -3623.559,E2 -3623.559} C_VEL
LIN {X 0,Y 545.08,Z 439.835,A -85,B 0,C 180,E1 -3626.001,E2 -3626.001} C_VEL
LIN {X 0,Y 545.084,Z 439.823,A -85,B 0,C 180,E1 -3628.749,E2 -3628.749} C_VEL
LIN {X 0,Y 545.07,Z 439.837,A -85,B 0,C 180,E1 -3631.683,E2 -3631.683} C_VEL
LIN {X 0,Y 545.073,Z 439.828,A -85,B 0,C 180,E1 -3634.564,E2 -3634.564} C_VEL
LIN {X 0,Y 545.035,Z 439.838,A -85,B 0,C 180,E1 -3637.304,E2 -3637.304} C_VEL
LIN {X 0,Y 545.087,Z 439.833,A -85,B 0,C 180,E1 -3640.141,E2 -3640.141} C_VEL
LIN {X 0,Y 545.08,Z 439.831,A -85,B 0,C 180,E1 -3643.106,E2 -3643.106} C_VEL
LIN {X 0,Y 545.05,Z 439.845,A -85,B 0,C 180,E1 -3646.226,E2 -3646.226} C_VEL
LIN {X 0,Y 545.092,Z 439.835,A -85,B 0,C 180,E1 -3648.888,E2 -3648.888} C_VEL
LIN {X 0,Y 545.048,Z 439.826,A -85,B 0,C 180,E1 -3651.763,E2 -3651.763} C_VEL
LIN {X 0,Y 545.061,Z 439.84,A -85,B 0,C 180,E1 -3654.534,E2 -3654.534} C_VEL
LIN {X 0,Y 545.12,Z 439.941,A -85,B 0,C 180,E1 -3657.709,E2 -3657.709} C_VEL
LIN {X 0,Y 545.816,Z 442.666,A -85,B 0,C 180,E1 -3658.192,E2 -3658.192} C_VEL
LIN {X 0,Y 548.299,Z 453.069,A -85,B 0,C 180,E1 -3659.833,E2 -3659.833} C_VEL
LIN {X 0,Y 547.66,Z 473.747,A -85,B 0,C 180,E1 -3662.693,E2 -3662.693} C_VEL
LIN {X 0,Y 547.405,Z 484.227,A -85,B 0,C 180,E1 -3664.094,E2 -3664.094} C_VEL
LIN {X 0,Y 550.653,Z 497.202,A -85,B 0,C 180,E1 -3664.466,E2 -3664.466} C_VEL
LIN {X 0,Y 549.667,Z 661.471,A -85,B 0,C 180,E1 -3666.727,E2 -3666.727} C_VEL
LIN {X 0,Y 549.379,Z 697.957,A -85,B 0,C 180,E1 -3667.252,E2 -3667.252} C_VEL
LIN {X 0,Y 549.147,Z 715.047,A -85,B 0,C 180,E1 -3667.646,E2 -3667.646} C_VEL
LIN {X 0,Y 548.728,Z 731.879,A -85,B 0,C 180,E1 -3668.197,E2 -3668.197} C_VEL
LIN {X 0,Y 548.326,Z 746.685,A -85,B 0,C 180,E1 -3668.821,E2 -3668.821} C_VEL
LIN {X 0,Y 547.903,Z 760.11,A -85,B 0,C 180,E1 -3669.51,E2 -3669.51} C_VEL
LIN {X 0,Y 547.377,Z 774.792,A -85,B 0,C 180,E1 -3670.402,E2 -3670.402} C_VEL
LIN {X 0,Y 546.856,Z 790.353,A -85,B 0,C 180,E1 -3671.551,E2 -3671.551} C_VEL
LIN {X 0,Y 546.381,Z 802.8,A -85,B 0,C 180,E1 -3672.634,E2 -3672.634} C_VEL
LIN {X 0,Y 546.005,Z 813.813,A -85,B 0,C 180,E1 -3673.743,E2 -3673.743} C_VEL
LIN {X 0,Y 545.641,Z 825.311,A -85,B 0,C 180,E1 -3675.072,E2 -3675.072} C_VEL
LIN {X 0,Y 545.321,Z 836.443,A -85,B 0,C 180,E1 -3676.587,E2 -3676.587} C_VEL
LIN {X 0,Y 545.08,Z 845.798,A -85,B 0,C 180,E1 -3678.095,E2 -3678.095} C_VEL
LIN {X 0,Y 544.905,Z 853.658,A -85,B 0,C 180,E1 -3679.597,E2 -3679.597} C_VEL
LIN {X 0,Y 544.768,Z 860.269,A -85,B 0,C 180,E1 -3681.094,E2 -3681.094} C_VEL
LIN {X 0,Y 544.712,Z 865.667,A -85,B 0,C 180,E1 -3682.587,E2 -3682.587} C_VEL
LIN {X 0,Y 544.686,Z 870.023,A -85,B 0,C 180,E1 -3684.075,E2 -3684.075} C_VEL
LIN {X 0,Y 544.597,Z 873.302,A -85,B 0,C 180,E1 -3685.559,E2 -3685.559} C_VEL
LIN {X 0,Y 544.64,Z 875.655,A -85,B 0,C 180,E1 -3687.041,E2 -3687.041} C_VEL
LIN {X 0,Y 544.539,Z 877.014,A -85,B 0,C 180,E1 -3688.521,E2 -3688.521} C_VEL
LIN {X 0,Y 544.536,Z 877.5,A -85,B 0,C 180,E1 -3690,E2 -3690} C_VEL
LIN {X 0,Y 544.539,Z 877.014,A -85,B 0,C 180,E1 -3691.479,E2 -3691.479} C_VEL
LIN {X 0,Y 544.64,Z 875.655,A -85,B 0,C 180,E1 -3692.959,E2 -3692.959} C_VEL
LIN {X 0,Y 544.597,Z 873.302,A -85,B 0,C 180,E1 -3694.441,E2 -3694.441} C_VEL
LIN {X 0,Y 544.686,Z 870.023,A -85,B 0,C 180,E1 -3695.925,E2 -3695.925} C_VEL
LIN {X 0,Y 544.712,Z 865.667,A -85,B 0,C 180,E1 -3697.413,E2 -3697.413} C_VEL
LIN {X 0,Y 544.768,Z 860.269,A -85,B 0,C 180,E1 -3698.906,E2 -3698.906} C_VEL
LIN {X 0,Y 544.906,Z 853.658,A -85,B 0,C 180,E1 -3700.403,E2 -3700.403} C_VEL
LIN {X 0,Y 545.076,Z 845.798,A -85,B 0,C 180,E1 -3701.905,E2 -3701.905} C_VEL
LIN {X 0,Y 545.321,Z 836.443,A -85,B 0,C 180,E1 -3703.413,E2 -3703.413} C_VEL
LIN {X 0,Y 545.668,Z 825.311,A -85,B 0,C 180,E1 -3704.927,E2 -3704.927} C_VEL
LIN {X 0,Y 546,Z 813.813,A -85,B 0,C 180,E1 -3706.258,E2 -3706.258} C_VEL
LIN {X 0,Y 546.461,Z 801.181,A -85,B 0,C 180,E1 -3707.519,E2 -3707.519} C_VEL
LIN {X 0,Y 546.997,Z 786.737,A -85,B 0,C 180,E1 -3708.736,E2 -3708.736} C_VEL
LIN {X 0,Y 547.448,Z 773.303,A -85,B 0,C 180,E1 -3709.693,E2 -3709.693} C_VEL
LIN {X 0,Y 547.866,Z 760.063,A -85,B 0,C 180,E1 -3710.494,E2 -3710.494} C_VEL
LIN {X 0,Y 548.312,Z 746.685,A -85,B 0,C 180,E1 -3711.179,E2 -3711.179} C_VEL
LIN {X 0,Y 548.72,Z 731.879,A -85,B 0,C 180,E1 -3711.803,E2 -3711.803} C_VEL
LIN {X 0,Y 549.124,Z 714.135,A -85,B 0,C 180,E1 -3712.38,E2 -3712.38} C_VEL
LIN {X 0,Y 549.427,Z 697.214,A -85,B 0,C 180,E1 -3712.759,E2 -3712.759} C_VEL
LIN {X 0,Y 549.749,Z 650.571,A -85,B 0,C 180,E1 -3713.422,E2 -3713.422} C_VEL
LIN {X 0,Y 550.587,Z 496.988,A -85,B 0,C 180,E1 -3715.54,E2 -3715.54} C_VEL
LIN {X 0,Y 547.443,Z 484.247,A -85,B 0,C 180,E1 -3715.902,E2 -3715.902} C_VEL
LIN {X 0,Y 547.906,Z 464.771,A -85,B 0,C 180,E1 -3718.541,E2 -3718.541} C_VEL
LIN {X 0,Y 548.244,Z 453.07,A -85,B 0,C 180,E1 -3720.17,E2 -3720.17} C_VEL
LIN {X 0,Y 546.876,Z 446.844,A -85,B 0,C 180,E1 -3721.144,E2 -3721.144} C_VEL
LIN {X 0,Y 545.134,Z 440.109,A -85,B 0,C 180,E1 -3722.236,E2 -3722.236} C_VEL
LIN {X 0,Y 545.067,Z 439.821,A -85,B 0,C 180,E1 -3723.671,E2 -3723.671} C_VEL
LIN {X 0,Y 545.051,Z 439.837,A -85,B 0,C 180,E1 -3726.379,E2 -3726.379} C_VEL
LIN {X 0,Y 545.1,Z 439.825,A -85,B 0,C 180,E1 -3729.324,E2 -3729.324} C_VEL
LIN {X 0,Y 545.074,Z 439.835,A -85,B 0,C 180,E1 -3732.102,E2 -3732.102} C_VEL
LIN {X 0,Y 545.057,Z 439.837,A -85,B 0,C 180,E1 -3735.166,E2 -3735.166} C_VEL
LIN {X 0,Y 545.077,Z 439.84,A -85,B 0,C 180,E1 -3737.897,E2 -3737.897} C_VEL
LIN {X 0,Y 545.1,Z 439.827,A -85,B 0,C 180,E1 -3740.675,E2 -3740.675} C_VEL
LIN {X 0,Y 545.054,Z 439.841,A -85,B 0,C 180,E1 -3743.621,E2 -3743.621} C_VEL
LIN {X 0,Y 545.063,Z 439.837,A -85,B 0,C 180,E1 -3746.328,E2 -3746.328} C_VEL
LIN {X 0,Y 545.062,Z 439.834,A -85,B 0,C 180,E1 -3748.952,E2 -3748.952} C_VEL
LIN {X 0,Y 545.096,Z 439.823,A -85,B 0,C 180,E1 -3751.507,E2 -3751.507} C_VEL
LIN {X 0,Y 545.091,Z 439.834,A -85,B 0,C 180,E1 -3754.49,E2 -3754.49} C_VEL
LIN {X 0,Y 545.036,Z 439.836,A -85,B 0,C 180,E1 -3757.242,E2 -3757.242} C_VEL
LIN {X 0,Y 545.112,Z 439.822,A -85,B 0,C 180,E1 -3760.415,E2 -3760.415} C_VEL
LIN {X 0,Y 545.066,Z 439.833,A -85,B 0,C 180,E1 -3763.521,E2 -3763.521} C_VEL
LIN {X 0,Y 545.086,Z 439.834,A -85,B 0,C 180,E1 -3765.82,E2 -3765.82} C_VEL
LIN {X 0,Y 545.123,Z 439.828,A -85,B 0,C 180,E1 -3768.849,E2 -3768.849} C_VEL
LIN {X 0,Y 545.125,Z 439.824,A -85,B 0,C 180,E1 -3771.847,E2 -3771.847} C_VEL
LIN {X 0,Y 545.2,Z 439.819,A -85,B 0,C 180,E1 -3774.823,E2 -3774.823} C_VEL
LIN {X 0,Y 545.186,Z 439.818,A -85,B 0,C 180,E1 -3777.784,E2 -3777.784} C_VEL
LIN {X 0,Y 545.207,Z 439.817,A -85,B 0,C 180,E1 -3780.738,E2 -3780.738} C_VEL
LIN {X 0,Y 545.168,Z 439.824,A -85,B 0,C 180,E1 -3782.956,E2 -3782.956} C_VEL
LIN {X 0,Y 545.169,Z 439.819,A -85,B 0,C 180,E1 -3785.919,E2 -3785.919} C_VEL
LIN {X 0,Y 545.119,Z 439.831,A -85,B 0,C 180,E1 -3788.9,E2 -3788.9} C_VEL
LIN {X 0,Y 545.126,Z 439.823,A -85,B 0,C 180,E1 -3791.904,E2 -3791.904} C_VEL
LIN {X 0,Y 545.075,Z 439.835,A -85,B 0,C 180,E1 -3794.944,E2 -3794.944} C_VEL
LIN {X 0,Y 545.073,Z 439.833,A -85,B 0,C 180,E1 -3798.026,E2 -3798.026} C_VEL
LIN {X 0,Y 545.089,Z 439.832,A -85,B 0,C 180,E1 -3800.372,E2 -3800.372} C_VEL
LIN {X 0,Y 545.082,Z 439.832,A -85,B 0,C 180,E1 -3803.559,E2 -3803.559} C_VEL
LIN {X 0,Y 545.079,Z 439.822,A -85,B 0,C 180,E1 -3806,E2 -3806} C_VEL
LIN {X 0,Y 545.083,Z 439.832,A -85,B 0,C 180,E1 -3808.749,E2 -3808.749} C_VEL
LIN {X 0,Y 545.069,Z 439.833,A -85,B 0,C 180,E1 -3811.683,E2 -3811.683} C_VEL
LIN {X 0,Y 545.072,Z 439.823,A -85,B 0,C 180,E1 -3814.563,E2 -3814.563} C_VEL
LIN {X 0,Y 545.063,Z 439.84,A -85,B 0,C 180,E1 -3817.019,E2 -3817.019} C_VEL
LIN {X 0,Y 544.388,Z 439.925,A -85,B 0,C 180,E1 -3817.635,E2 -3817.635} C_VEL
LIN {X 0,Y 541.533,Z 440.278,A -85,B 0,C 180,E1 -3818.636,E2 -3818.636} C_VEL
LIN {X 0,Y 539.133,Z 440.579,A -85,B 0,C 180,E1 -3819.442,E2 -3819.442} C_VEL
LIN {X 0,Y 538.117,Z 440.701,A -85,B 0,C 180,E1 -3820.064,E2 -3820.064} C_VEL
LIN {X 0,Y 538.041,Z 440.71,A -85,B 0,C 180,E1 -3820.274,E2 -3820.274} C_VEL
LIN {X 0,Y 538.025,Z 440.718,A -85,B 0,C 180,E1 -3822.989,E2 -3822.989} C_VEL
LIN {X 0,Y 538.022,Z 440.713,A -85,B 0,C 180,E1 -3825.926,E2 -3825.926} C_VEL
LIN {X 0,Y 538.071,Z 440.714,A -85,B 0,C 180,E1 -3829.249,E2 -3829.249} C_VEL
LIN {X 0,Y 537.987,Z 440.717,A -85,B 0,C 180,E1 -3832.123,E2 -3832.123} C_VEL
LIN {X 0,Y 538.015,Z 440.715,A -85,B 0,C 180,E1 -3834.918,E2 -3834.918} C_VEL
LIN {X 0,Y 538.026,Z 440.719,A -85,B 0,C 180,E1 -3837.619,E2 -3837.619} C_VEL
LIN {X 0,Y 538.013,Z 440.714,A -85,B 0,C 180,E1 -3840.239,E2 -3840.239} C_VEL
LIN {X 0,Y 538.066,Z 440.708,A -85,B 0,C 180,E1 -3842.797,E2 -3842.797} C_VEL
LIN {X 0,Y 538.045,Z 440.714,A -85,B 0,C 180,E1 -3845.293,E2 -3845.293} C_VEL
LIN {X 0,Y 538.011,Z 440.717,A -85,B 0,C 180,E1 -3848.042,E2 -3848.042} C_VEL
LIN {X 0,Y 538.036,Z 440.712,A -85,B 0,C 180,E1 -3850.94,E2 -3850.94} C_VEL
LIN {X 0,Y 538.023,Z 440.715,A -85,B 0,C 180,E1 -3853.299,E2 -3853.299} C_VEL
LIN {X 0,Y 538.061,Z 440.715,A -85,B 0,C 180,E1 -3855.631,E2 -3855.631} C_VEL
LIN {X 0,Y 538.073,Z 440.707,A -85,B 0,C 180,E1 -3858.702,E2 -3858.702} C_VEL
LIN {X 0,Y 538.083,Z 440.712,A -85,B 0,C 180,E1 -3861.74,E2 -3861.74} C_VEL
LIN {X 0,Y 538.157,Z 440.696,A -85,B 0,C 180,E1 -3864.755,E2 -3864.755} C_VEL
LIN {X 0,Y 538.166,Z 440.702,A -85,B 0,C 180,E1 -3867.755,E2 -3867.755} C_VEL
LIN {X 0,Y 538.178,Z 440.694,A -85,B 0,C 180,E1 -3870.748,E2 -3870.748} C_VEL
LIN {X 0,Y 538.136,Z 440.699,A -85,B 0,C 180,E1 -3872.994,E2 -3872.994} C_VEL
LIN {X 0,Y 538.12,Z 440.708,A -85,B 0,C 180,E1 -3875.997,E2 -3875.997} C_VEL
LIN {X 0,Y 538.065,Z 440.707,A -85,B 0,C 180,E1 -3879.017,E2 -3879.017} C_VEL
LIN {X 0,Y 538.08,Z 440.712,A -85,B 0,C 180,E1 -3882.062,E2 -3882.062} C_VEL
LIN {X 0,Y 538.042,Z 440.711,A -85,B 0,C 180,E1 -3885.143,E2 -3885.143} C_VEL
LIN {X 0,Y 538.031,Z 440.719,A -85,B 0,C 180,E1 -3888.27,E2 -3888.27} C_VEL
LIN {X 0,Y 538.035,Z 440.715,A -85,B 0,C 180,E1 -3890.651,E2 -3890.651} C_VEL
LIN {X 0,Y 537.999,Z 440.718,A -85,B 0,C 180,E1 -3893.888,E2 -3893.888} C_VEL
LIN {X 0,Y 538.045,Z 440.717,A -85,B 0,C 180,E1 -3896.366,E2 -3896.366} C_VEL
LIN {X 0,Y 538.026,Z 440.715,A -85,B 0,C 180,E1 -3898.933,E2 -3898.933} C_VEL
LIN {X 0,Y 538.022,Z 440.713,A -85,B 0,C 180,E1 -3901.89,E2 -3901.89} C_VEL
LIN {X 0,Y 538.029,Z 440.72,A -85,B 0,C 180,E1 -3904.621,E2 -3904.621} C_VEL
LIN {X 0,Y 538.001,Z 440.717,A -85,B 0,C 180,E1 -3907.17,E2 -3907.17} C_VEL
LIN {X 0,Y 538.047,Z 440.709,A -85,B 0,C 180,E1 -3909.794,E2 -3909.794} C_VEL
LIN {X 0,Y 538.012,Z 440.721,A -85,B 0,C 180,E1 -3912.785,E2 -3912.785} C_VEL
LIN {X 0,Y 538.024,Z 440.716,A -85,B 0,C 180,E1 -3915.14,E2 -3915.14} C_VEL
LIN {X 0,Y 538.051,Z 440.71,A -85,B 0,C 180,E1 -3918.229,E2 -3918.229} C_VEL
LIN {X 0,Y 538.008,Z 440.719,A -85,B 0,C 180,E1 -3921.17,E2 -3921.17} C_VEL
LIN {X 0,Y 538.021,Z 440.71,A -85,B 0,C 180,E1 -3924.083,E2 -3924.083} C_VEL
LIN {X 0,Y 538.022,Z 440.704,A -85,B 0,C 180,E1 -3926.727,E2 -3926.727} C_VEL
LIN {X 0,Y 538.029,Z 440.713,A -85,B 0,C 180,E1 -3929.554,E2 -3929.554} C_VEL
LIN {X 0,Y 538.039,Z 440.702,A -85,B 0,C 180,E1 -3931.95,E2 -3931.95} C_VEL
LIN {X 0,Y 538.066,Z 440.696,A -85,B 0,C 180,E1 -3934.467,E2 -3934.467} C_VEL
LIN {X 0,Y 538.014,Z 440.718,A -85,B 0,C 180,E1 -3936.928,E2 -3936.928} C_VEL
LIN {X 0,Y 538.069,Z 440.703,A -85,B 0,C 180,E1 -3940.148,E2 -3940.148} C_VEL
LIN {X 0,Y 538.017,Z 440.716,A -85,B 0,C 180,E1 -3943.299,E2 -3943.299} C_VEL
LIN {X 0,Y 538.054,Z 440.711,A -85,B 0,C 180,E1 -3945.631,E2 -3945.631} C_VEL
LIN {X 0,Y 538.08,Z 440.702,A -85,B 0,C 180,E1 -3948.702,E2 -3948.702} C_VEL
LIN {X 0,Y 538.081,Z 440.706,A -85,B 0,C 180,E1 -3951.74,E2 -3951.74} C_VEL
LIN {X 0,Y 538.178,Z 440.69,A -85,B 0,C 180,E1 -3954.755,E2 -3954.755} C_VEL
LIN {X 0,Y 538.158,Z 440.695,A -85,B 0,C 180,E1 -3957.755,E2 -3957.755} C_VEL
LIN {X 0,Y 538.176,Z 440.692,A -85,B 0,C 180,E1 -3960.748,E2 -3960.748} C_VEL
LIN {X 0,Y 538.134,Z 440.698,A -85,B 0,C 180,E1 -3962.995,E2 -3962.995} C_VEL
LIN {X 0,Y 538.115,Z 440.703,A -85,B 0,C 180,E1 -3965.998,E2 -3965.998} C_VEL
LIN {X 0,Y 538.068,Z 440.701,A -85,B 0,C 180,E1 -3969.018,E2 -3969.018} C_VEL
LIN {X 0,Y 538.075,Z 440.706,A -85,B 0,C 180,E1 -3972.063,E2 -3972.063} C_VEL
LIN {X 0,Y 538.036,Z 440.71,A -85,B 0,C 180,E1 -3975.144,E2 -3975.144} C_VEL
LIN {X 0,Y 538.026,Z 440.704,A -85,B 0,C 180,E1 -3978.27,E2 -3978.27} C_VEL
LIN {X 0,Y 538.033,Z 440.698,A -85,B 0,C 180,E1 -3980.652,E2 -3980.652} C_VEL
LIN {X 0,Y 538.015,Z 440.72,A -85,B 0,C 180,E1 -3983.888,E2 -3983.888} C_VEL
LIN {X 0,Y 538.041,Z 440.706,A -85,B 0,C 180,E1 -3986.367,E2 -3986.367} C_VEL
LIN {X 0,Y 538.029,Z 440.7,A -85,B 0,C 180,E1 -3988.935,E2 -3988.935} C_VEL
LIN {X 0,Y 538.02,Z 440.718,A -85,B 0,C 180,E1 -3991.891,E2 -3991.891} C_VEL
LIN {X 0,Y 538.023,Z 440.705,A -85,B 0,C 180,E1 -3994.621,E2 -3994.621} C_VEL
LIN {X 0,Y 538.004,Z 440.714,A -85,B 0,C 180,E1 -3997.172,E2 -3997.172} C_VEL
LIN {X 0,Y 538.048,Z 440.709,A -85,B 0,C 180,E1 -3999.795,E2 -3999.795} C_VEL
LIN {X 0,Y 538.017,Z 440.713,A -85,B 0,C 180,E1 -4002.786,E2 -4002.786} C_VEL
LIN {X 0,Y 538.026,Z 440.711,A -85,B 0,C 180,E1 -4005.141,E2 -4005.141} C_VEL
LIN {X 0,Y 538.035,Z 440.713,A -85,B 0,C 180,E1 -4008.228,E2 -4008.228} C_VEL
LIN {X 0,Y 538.01,Z 440.703,A -85,B 0,C 180,E1 -4011.17,E2 -4011.17} C_VEL
LIN {X 0,Y 538.026,Z 440.717,A -85,B 0,C 180,E1 -4014.084,E2 -4014.084} C_VEL
LIN {X 0,Y 538.039,Z 440.717,A -85,B 0,C 180,E1 -4017.287,E2 -4017.287} C_VEL
LIN {X 0,Y 538.146,Z 441.296,A -85,B 0,C 180,E1 -4017.516,E2 -4017.516} C_VEL
LIN {X 0,Y 541.5,Z 454.299,A -85,B 0,C 180,E1 -4019.592,E2 -4019.592} C_VEL
LIN {X 0,Y 541.036,Z 471.714,A -85,B 0,C 180,E1 -4022.044,E2 -4022.044} C_VEL
LIN {X 0,Y 540.69,Z 484.255,A -85,B 0,C 180,E1 -4023.75,E2 -4023.75} C_VEL
LIN {X 0,Y 544.247,Z 498.625,A -85,B 0,C 180,E1 -4024.164,E2 -4024.164} C_VEL
LIN {X 0,Y 543.153,Z 661.649,A -85,B 0,C 180,E1 -4026.433,E2 -4026.433} C_VEL
LIN {X 0,Y 542.85,Z 697.92,A -85,B 0,C 180,E1 -4026.963,E2 -4026.963} C_VEL
LIN {X 0,Y 542.534,Z 715.057,A -85,B 0,C 180,E1 -4027.358,E2 -4027.358} C_VEL
LIN {X 0,Y 542.113,Z 731.864,A -85,B 0,C 180,E1 -4027.917,E2 -4027.917} C_VEL
LIN {X 0,Y 541.656,Z 746.672,A -85,B 0,C 180,E1 -4028.548,E2 -4028.548} C_VEL
LIN {X 0,Y 541.21,Z 759.718,A -85,B 0,C 180,E1 -4029.223,E2 -4029.223} C_VEL
LIN {X 0,Y 540.712,Z 773.293,A -85,B 0,C 180,E1 -4030.051,E2 -4030.051} C_VEL
LIN {X 0,Y 540.148,Z 788.01,A -85,B 0,C 180,E1 -4031.116,E2 -4031.116} C_VEL
LIN {X 0,Y 539.613,Z 801.509,A -85,B 0,C 180,E1 -4032.284,E2 -4032.284} C_VEL
LIN {X 0,Y 539.086,Z 813.808,A -85,B 0,C 180,E1 -4033.528,E2 -4033.528} C_VEL
LIN {X 0,Y 538.68,Z 825.305,A -85,B 0,C 180,E1 -4034.875,E2 -4034.875} C_VEL
LIN {X 0,Y 538.317,Z 836.445,A -85,B 0,C 180,E1 -4036.409,E2 -4036.409} C_VEL
LIN {X 0,Y 538.029,Z 845.793,A -85,B 0,C 180,E1 -4037.937,E2 -4037.937} C_VEL
LIN {X 0,Y 537.858,Z 853.654,A -85,B 0,C 180,E1 -4039.46,E2 -4039.46} C_VEL
LIN {X 0,Y 537.69,Z 860.264,A -85,B 0,C 180,E1 -4040.976,E2 -4040.976} C_VEL
LIN {X 0,Y 537.634,Z 865.667,A -85,B 0,C 180,E1 -4042.489,E2 -4042.489} C_VEL
LIN {X 0,Y 537.587,Z 870.019,A -85,B 0,C 180,E1 -4043.997,E2 -4043.997} C_VEL
LIN {X 0,Y 537.497,Z 873.304,A -85,B 0,C 180,E1 -4045.5,E2 -4045.5} C_VEL
LIN {X 0,Y 537.54,Z 875.655,A -85,B 0,C 180,E1 -4047.002,E2 -4047.002} C_VEL
LIN {X 0,Y 537.444,Z 877.016,A -85,B 0,C 180,E1 -4048.501,E2 -4048.501} C_VEL
LIN {X 0,Y 537.437,Z 877.5,A -85,B 0,C 180,E1 -4050,E2 -4050} C_VEL
LIN {X 0,Y 537.444,Z 877.016,A -85,B 0,C 180,E1 -4051.499,E2 -4051.499} C_VEL
LIN {X 0,Y 537.54,Z 875.655,A -85,B 0,C 180,E1 -4052.998,E2 -4052.998} C_VEL
LIN {X 0,Y 537.497,Z 873.304,A -85,B 0,C 180,E1 -4054.5,E2 -4054.5} C_VEL
LIN {X 0,Y 537.587,Z 870.019,A -85,B 0,C 180,E1 -4056.003,E2 -4056.003} C_VEL
LIN {X 0,Y 537.634,Z 865.667,A -85,B 0,C 180,E1 -4057.511,E2 -4057.511} C_VEL
LIN {X 0,Y 537.69,Z 860.264,A -85,B 0,C 180,E1 -4059.024,E2 -4059.024} C_VEL
LIN {X 0,Y 537.858,Z 853.654,A -85,B 0,C 180,E1 -4060.54,E2 -4060.54} C_VEL
LIN {X 0,Y 538.028,Z 845.793,A -85,B 0,C 180,E1 -4062.063,E2 -4062.063} C_VEL
LIN {X 0,Y 538.317,Z 836.445,A -85,B 0,C 180,E1 -4063.591,E2 -4063.591} C_VEL
LIN {X 0,Y 538.729,Z 825.305,A -85,B 0,C 180,E1 -4065.124,E2 -4065.124} C_VEL
LIN {X 0,Y 539.085,Z 813.808,A -85,B 0,C 180,E1 -4066.472,E2 -4066.472} C_VEL
LIN {X 0,Y 539.584,Z 801.524,A -85,B 0,C 180,E1 -4067.716,E2 -4067.716} C_VEL
LIN {X 0,Y 540.194,Z 786.737,A -85,B 0,C 180,E1 -4068.98,E2 -4068.98} C_VEL
LIN {X 0,Y 540.708,Z 773.293,A -85,B 0,C 180,E1 -4069.949,E2 -4069.949} C_VEL
LIN {X 0,Y 541.196,Z 759.799,A -85,B 0,C 180,E1 -4070.773,E2 -4070.773} C_VEL
LIN {X 0,Y 541.642,Z 746.672,A -85,B 0,C 180,E1 -4071.453,E2 -4071.453} C_VEL
LIN {X 0,Y 542.081,Z 733.095,A -85,B 0,C 180,E1 -4072.034,E2 -4072.034} C_VEL
LIN {X 0,Y 542.497,Z 717.465,A -85,B 0,C 180,E1 -4072.568,E2 -4072.568} C_VEL
LIN {X 0,Y 542.849,Z 699.322,A -85,B 0,C 180,E1 -4073.012,E2 -4073.012} C_VEL
LIN {X 0,Y 543.08,Z 668.884,A -85,B 0,C 180,E1 -4073.468,E2 -4073.468} C_VEL
LIN {X 0,Y 544.16,Z 514.861,A -85,B 0,C 180,E1 -4075.607,E2 -4075.607} C_VEL
LIN {X 0,Y 544.223,Z 498.493,A -85,B 0,C 180,E1 -4075.839,E2 -4075.839} C_VEL
LIN {X 0,Y 540.68,Z 484.274,A -85,B 0,C 180,E1 -4076.248,E2 -4076.248} C_VEL
LIN {X 0,Y 541.185,Z 466.267,A -85,B 0,C 180,E1 -4078.717,E2 -4078.717} C_VEL
LIN {X 0,Y 541.501,Z 454.299,A -85,B 0,C 180,E1 -4080.408,E2 -4080.408} C_VEL
LIN {X 0,Y 538.055,Z 440.887,A -85,B 0,C 180,E1 -4082.574,E2 -4082.574} C_VEL
LIN {X 0,Y 538.016,Z 440.712,A -85,B 0,C 180,E1 -4085.082,E2 -4085.082} C_VEL
LIN {X 0,Y 537.988,Z 440.703,A -85,B 0,C 180,E1 -4087.877,E2 -4087.877} C_VEL
LIN {X 0,Y 538.046,Z 440.711,A -85,B 0,C 180,E1 -4090.775,E2 -4090.775} C_VEL
LIN {X 0,Y 538.018,Z 440.717,A -85,B 0,C 180,E1 -4094.073,E2 -4094.073} C_VEL
LIN {X 0,Y 538.027,Z 440.711,A -85,B 0,C 180,E1 -4097.011,E2 -4097.011} C_VEL
LIN {X 0,Y 538.072,Z 440.706,A -85,B 0,C 180,E1 -4099.248,E2 -4099.248} C_VEL
LIN {X 0,Y 537.989,Z 440.721,A -85,B 0,C 180,E1 -4102.122,E2 -4102.122} C_VEL
LIN {X 0,Y 538.012,Z 440.704,A -85,B 0,C 180,E1 -4104.917,E2 -4104.917} C_VEL
LIN {X 0,Y 538.024,Z 440.715,A -85,B 0,C 180,E1 -4107.618,E2 -4107.618} C_VEL
LIN {X 0,Y 538.035,Z 440.705,A -85,B 0,C 180,E1 -4110.24,E2 -4110.24} C_VEL
LIN {X 0,Y 538.063,Z 440.7,A -85,B 0,C 180,E1 -4112.796,E2 -4112.796} C_VEL
LIN {X 0,Y 538.041,Z 440.709,A -85,B 0,C 180,E1 -4115.292,E2 -4115.292} C_VEL
LIN {X 0,Y 538.006,Z 440.713,A -85,B 0,C 180,E1 -4118.041,E2 -4118.041} C_VEL
LIN {X 0,Y 538.031,Z 440.701,A -85,B 0,C 180,E1 -4120.94,E2 -4120.94} C_VEL
LIN {X 0,Y 538.017,Z 440.71,A -85,B 0,C 180,E1 -4123.299,E2 -4123.299} C_VEL
LIN {X 0,Y 538.054,Z 440.708,A -85,B 0,C 180,E1 -4125.63,E2 -4125.63} C_VEL
LIN {X 0,Y 538.08,Z 440.707,A -85,B 0,C 180,E1 -4128.702,E2 -4128.702} C_VEL
LIN {X 0,Y 538.081,Z 440.7,A -85,B 0,C 180,E1 -4131.739,E2 -4131.739} C_VEL
LIN {X 0,Y 538.157,Z 440.697,A -85,B 0,C 180,E1 -4134.755,E2 -4134.755} C_VEL
LIN {X 0,Y 538.158,Z 440.693,A -85,B 0,C 180,E1 -4137.755,E2 -4137.755} C_VEL
LIN {X 0,Y 538.176,Z 440.692,A -85,B 0,C 180,E1 -4140.748,E2 -4140.748} C_VEL
LIN {X 0,Y 538.134,Z 440.699,A -85,B 0,C 180,E1 -4142.994,E2 -4142.994} C_VEL
LIN {X 0,Y 538.123,Z 440.697,A -85,B 0,C 180,E1 -4145.997,E2 -4145.997} C_VEL
LIN {X 0,Y 538.068,Z 440.708,A -85,B 0,C 180,E1 -4149.017,E2 -4149.017} C_VEL
LIN {X 0,Y 538.074,Z 440.702,A -85,B 0,C 180,E1 -4152.062,E2 -4152.062} C_VEL
LIN {X 0,Y 538.035,Z 440.709,A -85,B 0,C 180,E1 -4155.144,E2 -4155.144} C_VEL
LIN {X 0,Y 538.026,Z 440.713,A -85,B 0,C 180,E1 -4158.27,E2 -4158.27} C_VEL
LIN {X 0,Y 538.033,Z 440.714,A -85,B 0,C 180,E1 -4160.651,E2 -4160.651} C_VEL
LIN {X 0,Y 538.014,Z 440.711,A -85,B 0,C 180,E1 -4163.888,E2 -4163.888} C_VEL
LIN {X 0,Y 538.041,Z 440.7,A -85,B 0,C 180,E1 -4166.366,E2 -4166.366} C_VEL
LIN {X 0,Y 538.047,Z 440.711,A -85,B 0,C 180,E1 -4168.939,E2 -4168.939} C_VEL
LIN {X 0,Y 538.018,Z 440.71,A -85,B 0,C 180,E1 -4171.891,E2 -4171.891} C_VEL
LIN {X 0,Y 538.022,Z 440.701,A -85,B 0,C 180,E1 -4174.621,E2 -4174.621} C_VEL
LIN {X 0,Y 538.015,Z 440.721,A -85,B 0,C 180,E1 -4177.173,E2 -4177.173} C_VEL
LIN {X 0,Y 538.041,Z 440.71,A -85,B 0,C 180,E1 -4180.274,E2 -4180.274} C_VEL
LIN {X 0,Y 537.39,Z 440.797,A -85,B 0,C 180,E1 -4180.9,E2 -4180.9} C_VEL
LIN {X 0,Y 534.53,Z 441.157,A -85,B 0,C 180,E1 -4181.914,E2 -4181.914} C_VEL
LIN {X 0,Y 532.096,Z 441.461,A -85,B 0,C 180,E1 -4182.731,E2 -4182.731} C_VEL
LIN {X 0,Y 531.044,Z 441.589,A -85,B 0,C 180,E1 -4183.362,E2 -4183.362} C_VEL
LIN {X 0,Y 530.955,Z 441.597,A -85,B 0,C 180,E1 -4183.576,E2 -4183.576} C_VEL
LIN {X 0,Y 530.957,Z 441.593,A -85,B 0,C 180,E1 -4186.506,E2 -4186.506} C_VEL
LIN {X 0,Y 531.019,Z 441.59,A -85,B 0,C 180,E1 -4189.572,E2 -4189.572} C_VEL
LIN {X 0,Y 530.962,Z 441.592,A -85,B 0,C 180,E1 -4192.577,E2 -4192.577} C_VEL
LIN {X 0,Y 530.998,Z 441.595,A -85,B 0,C 180,E1 -4195.312,E2 -4195.312} C_VEL
LIN {X 0,Y 530.977,Z 441.592,A -85,B 0,C 180,E1 -4198.033,E2 -4198.033} C_VEL
LIN {X 0,Y 530.984,Z 441.591,A -85,B 0,C 180,E1 -4200.874,E2 -4200.874} C_VEL
LIN {X 0,Y 531.007,Z 441.592,A -85,B 0,C 180,E1 -4203.257,E2 -4203.257} C_VEL
LIN {X 0,Y 530.992,Z 441.593,A -85,B 0,C 180,E1 -4205.958,E2 -4205.958} C_VEL
LIN {X 0,Y 530.995,Z 441.589,A -85,B 0,C 180,E1 -4209.062,E2 -4209.062} C_VEL
LIN {X 0,Y 531.013,Z 441.587,A -85,B 0,C 180,E1 -4212.278,E2 -4212.278} C_VEL
LIN {X 0,Y 531.016,Z 441.591,A -85,B 0,C 180,E1 -4215.436,E2 -4215.436} C_VEL
LIN {X 0,Y 531.045,Z 441.583,A -85,B 0,C 180,E1 -4218.55,E2 -4218.55} C_VEL
LIN {X 0,Y 531.052,Z 441.586,A -85,B 0,C 180,E1 -4221.63,E2 -4221.63} C_VEL
LIN {X 0,Y 531.117,Z 441.574,A -85,B 0,C 180,E1 -4224.685,E2 -4224.685} C_VEL
LIN {X 0,Y 531.137,Z 441.577,A -85,B 0,C 180,E1 -4227.725,E2 -4227.725} C_VEL
LIN {X 0,Y 531.149,Z 441.57,A -85,B 0,C 180,E1 -4230.758,E2 -4230.758} C_VEL
LIN {X 0,Y 531.103,Z 441.575,A -85,B 0,C 180,E1 -4233.034,E2 -4233.034} C_VEL
LIN {X 0,Y 531.08,Z 441.584,A -85,B 0,C 180,E1 -4236.077,E2 -4236.077} C_VEL
LIN {X 0,Y 531.026,Z 441.584,A -85,B 0,C 180,E1 -4239.138,E2 -4239.138} C_VEL
LIN {X 0,Y 531.037,Z 441.591,A -85,B 0,C 180,E1 -4242.225,E2 -4242.225} C_VEL
LIN {X 0,Y 530.992,Z 441.589,A -85,B 0,C 180,E1 -4245.349,E2 -4245.349} C_VEL
LIN {X 0,Y 531.013,Z 441.587,A -85,B 0,C 180,E1 -4247.722,E2 -4247.722} C_VEL
LIN {X 0,Y 530.995,Z 441.589,A -85,B 0,C 180,E1 -4250.938,E2 -4250.938} C_VEL
LIN {X 0,Y 530.967,Z 441.598,A -85,B 0,C 180,E1 -4254.225,E2 -4254.225} C_VEL
LIN {X 0,Y 531.007,Z 441.592,A -85,B 0,C 180,E1 -4256.743,E2 -4256.743} C_VEL
LIN {X 0,Y 530.977,Z 441.591,A -85,B 0,C 180,E1 -4259.322,E2 -4259.322} C_VEL
LIN {X 0,Y 530.974,Z 441.593,A -85,B 0,C 180,E1 -4262.103,E2 -4262.103} C_VEL
LIN {X 0,Y 530.985,Z 441.594,A -85,B 0,C 180,E1 -4264.854,E2 -4264.854} C_VEL
LIN {X 0,Y 530.96,Z 441.593,A -85,B 0,C 180,E1 -4267.507,E2 -4267.507} C_VEL
LIN {X 0,Y 531.019,Z 441.59,A -85,B 0,C 180,E1 -4270.428,E2 -4270.428} C_VEL
LIN {X 0,Y 530.957,Z 441.593,A -85,B 0,C 180,E1 -4273.494,E2 -4273.494} C_VEL
LIN {X 0,Y 530.958,Z 441.598,A -85,B 0,C 180,E1 -4276.505,E2 -4276.505} C_VEL
LIN {X 0,Y 531.002,Z 441.587,A -85,B 0,C 180,E1 -4279.569,E2 -4279.569} C_VEL
LIN {X 0,Y 530.968,Z 441.596,A -85,B 0,C 180,E1 -4282.575,E2 -4282.575} C_VEL
LIN {X 0,Y 530.992,Z 441.576,A -85,B 0,C 180,E1 -4285.311,E2 -4285.311} C_VEL
LIN {X 0,Y 530.973,Z 441.587,A -85,B 0,C 180,E1 -4288.033,E2 -4288.033} C_VEL
LIN {X 0,Y 530.998,Z 441.593,A -85,B 0,C 180,E1 -4290.87,E2 -4290.87} C_VEL
LIN {X 0,Y 531.002,Z 441.576,A -85,B 0,C 180,E1 -4293.257,E2 -4293.257} C_VEL
LIN {X 0,Y 530.987,Z 441.586,A -85,B 0,C 180,E1 -4295.957,E2 -4295.957} C_VEL
LIN {X 0,Y 530.992,Z 441.592,A -85,B 0,C 180,E1 -4299.062,E2 -4299.062} C_VEL
LIN {X 0,Y 531.007,Z 441.585,A -85,B 0,C 180,E1 -4302.278,E2 -4302.278} C_VEL
LIN {X 0,Y 531.03,Z 441.589,A -85,B 0,C 180,E1 -4305.436,E2 -4305.436} C_VEL
LIN {X 0,Y 531.037,Z 441.578,A -85,B 0,C 180,E1 -4308.55,E2 -4308.55} C_VEL
LIN {X 0,Y 531.05,Z 441.583,A -85,B 0,C 180,E1 -4311.63,E2 -4311.63} C_VEL
LIN {X 0,Y 531.134,Z 441.567,A -85,B 0,C 180,E1 -4314.686,E2 -4314.686} C_VEL
LIN {X 0,Y 531.13,Z 441.57,A -85,B 0,C 180,E1 -4317.725,E2 -4317.725} C_VEL
LIN {X 0,Y 531.146,Z 441.568,A -85,B 0,C 180,E1 -4320.758,E2 -4320.758} C_VEL
LIN {X 0,Y 531.101,Z 441.574,A -85,B 0,C 180,E1 -4323.034,E2 -4323.034} C_VEL
LIN {X 0,Y 531.074,Z 441.579,A -85,B 0,C 180,E1 -4326.077,E2 -4326.077} C_VEL
LIN {X 0,Y 531.027,Z 441.579,A -85,B 0,C 180,E1 -4329.138,E2 -4329.138} C_VEL
LIN {X 0,Y 531.032,Z 441.581,A -85,B 0,C 180,E1 -4332.225,E2 -4332.225} C_VEL
LIN {X 0,Y 530.987,Z 441.59,A -85,B 0,C 180,E1 -4335.35,E2 -4335.35} C_VEL
LIN {X 0,Y 531.007,Z 441.587,A -85,B 0,C 180,E1 -4337.723,E2 -4337.723} C_VEL
LIN {X 0,Y 530.993,Z 441.573,A -85,B 0,C 180,E1 -4340.938,E2 -4340.938} C_VEL
LIN {X 0,Y 530.971,Z 441.595,A -85,B 0,C 180,E1 -4344.225,E2 -4344.225} C_VEL
LIN {X 0,Y 531.003,Z 441.579,A -85,B 0,C 180,E1 -4346.744,E2 -4346.744} C_VEL
LIN {X 0,Y 530.985,Z 441.577,A -85,B 0,C 180,E1 -4349.322,E2 -4349.322} C_VEL
LIN {X 0,Y 530.973,Z 441.598,A -85,B 0,C 180,E1 -4352.104,E2 -4352.104} C_VEL
LIN {X 0,Y 530.981,Z 441.58,A -85,B 0,C 180,E1 -4354.855,E2 -4354.855} C_VEL
LIN {X 0,Y 530.961,Z 441.593,A -85,B 0,C 180,E1 -4357.508,E2 -4357.508} C_VEL
LIN {X 0,Y 531.02,Z 441.585,A -85,B 0,C 180,E1 -4360.429,E2 -4360.429} C_VEL
LIN {X 0,Y 530.96,Z 441.591,A -85,B 0,C 180,E1 -4363.495,E2 -4363.495} C_VEL
LIN {X 0,Y 530.953,Z 441.596,A -85,B 0,C 180,E1 -4366.505,E2 -4366.505} C_VEL
LIN {X 0,Y 530.984,Z 441.592,A -85,B 0,C 180,E1 -4368.976,E2 -4368.976} C_VEL
LIN {X 0,Y 530.953,Z 441.58,A -85,B 0,C 180,E1 -4371.53,E2 -4371.53} C_VEL
LIN {X 0,Y 530.978,Z 441.596,A -85,B 0,C 180,E1 -4374.383,E2 -4374.383} C_VEL
LIN {X 0,Y 531.015,Z 441.716,A -85,B 0,C 180,E1 -4377.085,E2 -4377.085} C_VEL
LIN {X 0,Y 532.652,Z 447.924,A -85,B 0,C 180,E1 -4378.146,E2 -4378.146} C_VEL
LIN {X 0,Y 534.83,Z 457.162,A -85,B 0,C 180,E1 -4379.609,E2 -4379.609} C_VEL
LIN {X 0,Y 534.145,Z 476.865,A -85,B 0,C 180,E1 -4382.386,E2 -4382.386} C_VEL
LIN {X 0,Y 533.968,Z 484.416,A -85,B 0,C 180,E1 -4383.404,E2 -4383.404} C_VEL
LIN {X 0,Y 537.883,Z 500.065,A -85,B 0,C 180,E1 -4383.857,E2 -4383.857} C_VEL
LIN {X 0,Y 536.624,Z 664.035,A -85,B 0,C 180,E1 -4386.163,E2 -4386.163} C_VEL
LIN {X 0,Y 536.314,Z 697.889,A -85,B 0,C 180,E1 -4386.666,E2 -4386.666} C_VEL
LIN {X 0,Y 535.992,Z 715.067,A -85,B 0,C 180,E1 -4387.066,E2 -4387.066} C_VEL
LIN {X 0,Y 535.524,Z 731.848,A -85,B 0,C 180,E1 -4387.631,E2 -4387.631} C_VEL
LIN {X 0,Y 535.055,Z 745.636,A -85,B 0,C 180,E1 -4388.219,E2 -4388.219} C_VEL
LIN {X 0,Y 534.628,Z 757.693,A -85,B 0,C 180,E1 -4388.838,E2 -4388.838} C_VEL
LIN {X 0,Y 534.129,Z 770.293,A -85,B 0,C 180,E1 -4389.594,E2 -4389.594} C_VEL
LIN {X 0,Y 533.559,Z 782.86,A -85,B 0,C 180,E1 -4390.474,E2 -4390.474} C_VEL
LIN {X 0,Y 533.055,Z 794.915,A -85,B 0,C 180,E1 -4391.454,E2 -4391.454} C_VEL
LIN {X 0,Y 532.42,Z 808.383,A -85,B 0,C 180,E1 -4392.723,E2 -4392.723} C_VEL
LIN {X 0,Y 531.927,Z 820.633,A -85,B 0,C 180,E1 -4394.089,E2 -4394.089} C_VEL
LIN {X 0,Y 531.586,Z 831.057,A -85,B 0,C 180,E1 -4395.452,E2 -4395.452} C_VEL
LIN {X 0,Y 531.205,Z 840.094,A -85,B 0,C 180,E1 -4396.808,E2 -4396.808} C_VEL
LIN {X 0,Y 530.965,Z 847.836,A -85,B 0,C 180,E1 -4398.154,E2 -4398.154} C_VEL
LIN {X 0,Y 530.766,Z 855.446,A -85,B 0,C 180,E1 -4399.703,E2 -4399.703} C_VEL
LIN {X 0,Y 530.594,Z 863.135,A -85,B 0,C 180,E1 -4401.622,E2 -4401.622} C_VEL
LIN {X 0,Y 530.546,Z 867.961,A -85,B 0,C 180,E1 -4403.153,E2 -4403.153} C_VEL
LIN {X 0,Y 530.468,Z 871.765,A -85,B 0,C 180,E1 -4404.679,E2 -4404.679} C_VEL
LIN {X 0,Y 530.477,Z 874.547,A -85,B 0,C 180,E1 -4406.202,E2 -4406.202} C_VEL
LIN {X 0,Y 530.404,Z 876.412,A -85,B 0,C 180,E1 -4407.722,E2 -4407.722} C_VEL
LIN {X 0,Y 530.339,Z 877.326,A -85,B 0,C 180,E1 -4409.241,E2 -4409.241} C_VEL
LIN {X 0,Y 530.339,Z 877.326,A -85,B 0,C 180,E1 -4410.759,E2 -4410.759} C_VEL
LIN {X 0,Y 530.404,Z 876.412,A -85,B 0,C 180,E1 -4412.278,E2 -4412.278} C_VEL
LIN {X 0,Y 530.477,Z 874.547,A -85,B 0,C 180,E1 -4413.798,E2 -4413.798} C_VEL
LIN {X 0,Y 530.468,Z 871.765,A -85,B 0,C 180,E1 -4415.321,E2 -4415.321} C_VEL
LIN {X 0,Y 530.56,Z 866.895,A -85,B 0,C 180,E1 -4417.229,E2 -4417.229} C_VEL
LIN {X 0,Y 530.612,Z 861.745,A -85,B 0,C 180,E1 -4418.761,E2 -4418.761} C_VEL
LIN {X 0,Y 530.766,Z 855.446,A -85,B 0,C 180,E1 -4420.297,E2 -4420.297} C_VEL
LIN {X 0,Y 530.983,Z 846.832,A -85,B 0,C 180,E1 -4422.032,E2 -4422.032} C_VEL
LIN {X 0,Y 531.281,Z 837.686,A -85,B 0,C 180,E1 -4423.58,E2 -4423.58} C_VEL
LIN {X 0,Y 531.753,Z 825.949,A -85,B 0,C 180,E1 -4425.245,E2 -4425.245} C_VEL
LIN {X 0,Y 532.125,Z 815.567,A -85,B 0,C 180,E1 -4426.496,E2 -4426.496} C_VEL
LIN {X 0,Y 532.579,Z 804.424,A -85,B 0,C 180,E1 -4427.668,E2 -4427.668} C_VEL
LIN {X 0,Y 533.151,Z 792.639,A -85,B 0,C 180,E1 -4428.742,E2 -4428.742} C_VEL
LIN {X 0,Y 533.715,Z 778.961,A -85,B 0,C 180,E1 -4429.82,E2 -4429.82} C_VEL
LIN {X 0,Y 534.379,Z 762.414,A -85,B 0,C 180,E1 -4430.898,E2 -4430.898} C_VEL
LIN {X 0,Y 534.949,Z 748.705,A -85,B 0,C 180,E1 -4431.634,E2 -4431.634} C_VEL
LIN {X 0,Y 535.411,Z 735.543,A -85,B 0,C 180,E1 -4432.222,E2 -4432.222} C_VEL
LIN {X 0,Y 535.798,Z 722.043,A -85,B 0,C 180,E1 -4432.713,E2 -4432.713} C_VEL
LIN {X 0,Y 536.115,Z 708.289,A -85,B 0,C 180,E1 -4433.107,E2 -4433.107} C_VEL
LIN {X 0,Y 536.379,Z 694.051,A -85,B 0,C 180,E1 -4433.401,E2 -4433.401} C_VEL
LIN {X 0,Y 537.702,Z 524.458,A -85,B 0,C 180,E1 -4435.798,E2 -4435.798} C_VEL
LIN {X 0,Y 537.745,Z 499.627,A -85,B 0,C 180,E1 -4436.157,E2 -4436.157} C_VEL
LIN {X 0,Y 533.937,Z 484.194,A -85,B 0,C 180,E1 -4436.611,E2 -4436.611} C_VEL
LIN {X 0,Y 534.638,Z 463.713,A -85,B 0,C 180,E1 -4439.469,E2 -4439.469} C_VEL
LIN {X 0,Y 534.788,Z 457.161,A -85,B 0,C 180,E1 -4440.394,E2 -4440.394} C_VEL
LIN {X 0,Y 532.964,Z 449.315,A -85,B 0,C 180,E1 -4441.633,E2 -4441.633} C_VEL
LIN {X 0,Y 531.015,Z 441.701,A -85,B 0,C 180,E1 -4442.915,E2 -4442.915} C_VEL
LIN {X 0,Y 530.978,Z 441.597,A -85,B 0,C 180,E1 -4445.617,E2 -4445.617} C_VEL
LIN {X 0,Y 530.963,Z 441.58,A -85,B 0,C 180,E1 -4448.653,E2 -4448.653} C_VEL
LIN {X 0,Y 530.991,Z 441.595,A -85,B 0,C 180,E1 -4451.435,E2 -4451.435} C_VEL
LIN {X 0,Y 530.981,Z 441.589,A -85,B 0,C 180,E1 -4454.546,E2 -4454.546} C_VEL
LIN {X 0,Y 530.982,Z 441.597,A -85,B 0,C 180,E1 -4457.833,E2 -4457.833} C_VEL
LIN {X 0,Y 530.999,Z 441.584,A -85,B 0,C 180,E1 -4460.558,E2 -4460.558} C_VEL
LIN {X 0,Y 530.968,Z 441.592,A -85,B 0,C 180,E1 -4463.842,E2 -4463.842} C_VEL
LIN {X 0,Y 530.992,Z 441.588,A -85,B 0,C 180,E1 -4466.494,E2 -4466.494} C_VEL
LIN {X 0,Y 530.974,Z 441.59,A -85,B 0,C 180,E1 -4469.353,E2 -4469.353} C_VEL
LIN {X 0,Y 531.009,Z 441.581,A -85,B 0,C 180,E1 -4472.466,E2 -4472.466} C_VEL
LIN {X 0,Y 530.999,Z 441.586,A -85,B 0,C 180,E1 -4474.942,E2 -4474.942} C_VEL
LIN {X 0,Y 530.963,Z 441.585,A -85,B 0,C 180,E1 -4478.246,E2 -4478.246} C_VEL
LIN {X 0,Y 530.988,Z 441.579,A -85,B 0,C 180,E1 -4480.677,E2 -4480.677} C_VEL
LIN {X 0,Y 530.983,Z 441.587,A -85,B 0,C 180,E1 -4483.071,E2 -4483.071} C_VEL
LIN {X 0,Y 531.009,Z 441.584,A -85,B 0,C 180,E1 -4485.436,E2 -4485.436} C_VEL
LIN {X 0,Y 531.037,Z 441.587,A -85,B 0,C 180,E1 -4488.55,E2 -4488.55} C_VEL
LIN {X 0,Y 531.051,Z 441.575,A -85,B 0,C 180,E1 -4491.629,E2 -4491.629} C_VEL
LIN {X 0,Y 531.115,Z 441.575,A -85,B 0,C 180,E1 -4494.685,E2 -4494.685} C_VEL
LIN {X 0,Y 531.13,Z 441.568,A -85,B 0,C 180,E1 -4497.725,E2 -4497.725} C_VEL
LIN {X 0,Y 531.146,Z 441.567,A -85,B 0,C 180,E1 -4500.758,E2 -4500.758} C_VEL
LIN {X 0,Y 531.1,Z 441.575,A -85,B 0,C 180,E1 -4503.034,E2 -4503.034} C_VEL
LIN {X 0,Y 531.081,Z 441.575,A -85,B 0,C 180,E1 -4506.077,E2 -4506.077} C_VEL
LIN {X 0,Y 531.027,Z 441.584,A -85,B 0,C 180,E1 -4509.138,E2 -4509.138} C_VEL
LIN {X 0,Y 531.031,Z 441.581,A -85,B 0,C 180,E1 -4512.225,E2 -4512.225} C_VEL
LIN {X 0,Y 530.986,Z 441.584,A -85,B 0,C 180,E1 -4515.35,E2 -4515.35} C_VEL
LIN {X 0,Y 531.007,Z 441.585,A -85,B 0,C 180,E1 -4517.722,E2 -4517.722} C_VEL
LIN {X 0,Y 530.992,Z 441.593,A -85,B 0,C 180,E1 -4520.938,E2 -4520.938} C_VEL
LIN {X 0,Y 530.97,Z 441.589,A -85,B 0,C 180,E1 -4524.225,E2 -4524.225} C_VEL
LIN {X 0,Y 531.002,Z 441.576,A -85,B 0,C 180,E1 -4526.743,E2 -4526.743} C_VEL
LIN {X 0,Y 530.991,Z 441.592,A -85,B 0,C 180,E1 -4529.322,E2 -4529.322} C_VEL
LIN {X 0,Y 530.971,Z 441.588,A -85,B 0,C 180,E1 -4532.103,E2 -4532.103} C_VEL
LIN {X 0,Y 530.979,Z 441.58,A -85,B 0,C 180,E1 -4534.854,E2 -4534.854} C_VEL
LIN {X 0,Y 530.965,Z 441.595,A -85,B 0,C 180,E1 -4537.507,E2 -4537.507} C_VEL
LIN {X 0,Y 531.002,Z 441.587,A -85,B 0,C 180,E1 -4540.431,E2 -4540.431} C_VEL
LIN {X 0,Y 530.958,Z 441.598,A -85,B 0,C 180,E1 -4543.495,E2 -4543.495} C_VEL
LIN {X 0,Y 530.955,Z 441.597,A -85,B 0,C 180,E1 -4543.576,E2 -4543.576} C_VEL
LIN {X 0,Y 530.282,Z 441.678,A -85,B 0,C 180,E1 -4544.209,E2 -4544.209} C_VEL
LIN {X 0,Y 527.433,Z 442.039,A -85,B 0,C 180,E1 -4545.238,E2 -4545.238} C_VEL
LIN {X 0,Y 525.029,Z 442.338,A -85,B 0,C 180,E1 -4546.067,E2 -4546.067} C_VEL
LIN {X 0,Y 523.996,Z 442.463,A -85,B 0,C 180,E1 -4546.706,E2 -4546.706} C_VEL
LIN {X 0,Y 523.911,Z 442.473,A -85,B 0,C 180,E1 -4546.923,E2 -4546.923} C_VEL
LIN {X 0,Y 523.971,Z 442.464,A -85,B 0,C 180,E1 -4549.924,E2 -4549.924} C_VEL
LIN {X 0,Y 523.905,Z 442.474,A -85,B 0,C 180,E1 -4552.869,E2 -4552.869} C_VEL
LIN {X 0,Y 523.94,Z 442.472,A -85,B 0,C 180,E1 -4555.711,E2 -4555.711} C_VEL
LIN {X 0,Y 523.926,Z 442.469,A -85,B 0,C 180,E1 -4558.457,E2 -4558.457} C_VEL
LIN {X 0,Y 523.935,Z 442.471,A -85,B 0,C 180,E1 -4561.126,E2 -4561.126} C_VEL
LIN {X 0,Y 523.981,Z 442.465,A -85,B 0,C 180,E1 -4563.98,E2 -4563.98} C_VEL
LIN {X 0,Y 523.932,Z 442.469,A -85,B 0,C 180,E1 -4566.271,E2 -4566.271} C_VEL
LIN {X 0,Y 523.941,Z 442.466,A -85,B 0,C 180,E1 -4568.767,E2 -4568.767} C_VEL
LIN {X 0,Y 523.949,Z 442.47,A -85,B 0,C 180,E1 -4571.221,E2 -4571.221} C_VEL
LIN {X 0,Y 523.935,Z 442.475,A -85,B 0,C 180,E1 -4573.639,E2 -4573.639} C_VEL
LIN {X 0,Y 523.937,Z 442.473,A -85,B 0,C 180,E1 -4576.028,E2 -4576.028} C_VEL
LIN {X 0,Y 524.011,Z 442.461,A -85,B 0,C 180,E1 -4578.394,E2 -4578.394} C_VEL
LIN {X 0,Y 524,Z 442.464,A -85,B 0,C 180,E1 -4581.516,E2 -4581.516} C_VEL
LIN {X 0,Y 524.078,Z 442.451,A -85,B 0,C 180,E1 -4584.614,E2 -4584.614} C_VEL
LIN {X 0,Y 524.109,Z 442.452,A -85,B 0,C 180,E1 -4587.695,E2 -4587.695} C_VEL
LIN {X 0,Y 524.119,Z 442.446,A -85,B 0,C 180,E1 -4590.768,E2 -4590.768} C_VEL
LIN {X 0,Y 524.069,Z 442.452,A -85,B 0,C 180,E1 -4593.075,E2 -4593.075} C_VEL
LIN {X 0,Y 524.042,Z 442.461,A -85,B 0,C 180,E1 -4596.159,E2 -4596.159} C_VEL
LIN {X 0,Y 523.994,Z 442.461,A -85,B 0,C 180,E1 -4599.262,E2 -4599.262} C_VEL
LIN {X 0,Y 524.021,Z 442.461,A -85,B 0,C 180,E1 -4601.751,E2 -4601.751} C_VEL
LIN {X 0,Y 523.989,Z 442.462,A -85,B 0,C 180,E1 -4605.052,E2 -4605.052} C_VEL
LIN {X 0,Y 523.96,Z 442.468,A -85,B 0,C 180,E1 -4607.969,E2 -4607.969} C_VEL
LIN {X 0,Y 523.967,Z 442.471,A -85,B 0,C 180,E1 -4610.41,E2 -4610.41} C_VEL
LIN {X 0,Y 523.906,Z 442.474,A -85,B 0,C 180,E1 -4612.893,E2 -4612.893} C_VEL
LIN {X 0,Y 523.95,Z 442.466,A -85,B 0,C 180,E1 -4615.418,E2 -4615.418} C_VEL
LIN {X 0,Y 523.966,Z 442.467,A -85,B 0,C 180,E1 -4617.998,E2 -4617.998} C_VEL
LIN {X 0,Y 523.941,Z 442.471,A -85,B 0,C 180,E1 -4620.855,E2 -4620.855} C_VEL
LIN {X 0,Y 523.957,Z 442.465,A -85,B 0,C 180,E1 -4623.735,E2 -4623.735} C_VEL
LIN {X 0,Y 523.916,Z 442.475,A -85,B 0,C 180,E1 -4626.404,E2 -4626.404} C_VEL
LIN {X 0,Y 523.924,Z 442.472,A -85,B 0,C 180,E1 -4629.083,E2 -4629.083} C_VEL
LIN {X 0,Y 523.965,Z 442.465,A -85,B 0,C 180,E1 -4631.312,E2 -4631.312} C_VEL
LIN {X 0,Y 523.948,Z 442.473,A -85,B 0,C 180,E1 -4634.691,E2 -4634.691} C_VEL
LIN {X 0,Y 523.957,Z 442.465,A -85,B 0,C 180,E1 -4637.882,E2 -4637.882} C_VEL
LIN {X 0,Y 523.952,Z 442.473,A -85,B 0,C 180,E1 -4640.919,E2 -4640.919} C_VEL
LIN {X 0,Y 523.919,Z 442.467,A -85,B 0,C 180,E1 -4643.827,E2 -4643.827} C_VEL
LIN {X 0,Y 523.933,Z 442.455,A -85,B 0,C 180,E1 -4646.635,E2 -4646.635} C_VEL
LIN {X 0,Y 523.955,Z 442.468,A -85,B 0,C 180,E1 -4649.356,E2 -4649.356} C_VEL
LIN {X 0,Y 523.971,Z 442.454,A -85,B 0,C 180,E1 -4652.28,E2 -4652.28} C_VEL
LIN {X 0,Y 523.945,Z 442.454,A -85,B 0,C 180,E1 -4654.581,E2 -4654.581} C_VEL
LIN {X 0,Y 523.907,Z 442.478,A -85,B 0,C 180,E1 -4657.107,E2 -4657.107} C_VEL
LIN {X 0,Y 523.969,Z 442.46,A -85,B 0,C 180,E1 -4659.866,E2 -4659.866} C_VEL
LIN {X 0,Y 523.961,Z 442.467,A -85,B 0,C 180,E1 -4662.837,E2 -4662.837} C_VEL
LIN {X 0,Y 523.994,Z 442.463,A -85,B 0,C 180,E1 -4665.236,E2 -4665.236} C_VEL
LIN {X 0,Y 524.002,Z 442.454,A -85,B 0,C 180,E1 -4668.394,E2 -4668.394} C_VEL
LIN {X 0,Y 523.998,Z 442.464,A -85,B 0,C 180,E1 -4671.516,E2 -4671.516} C_VEL
LIN {X 0,Y 524.093,Z 442.444,A -85,B 0,C 180,E1 -4674.614,E2 -4674.614} C_VEL
LIN {X 0,Y 524.102,Z 442.446,A -85,B 0,C 180,E1 -4677.695,E2 -4677.695} C_VEL
LIN {X 0,Y 524.116,Z 442.444,A -85,B 0,C 180,E1 -4680.768,E2 -4680.768} C_VEL
LIN {X 0,Y 524.067,Z 442.451,A -85,B 0,C 180,E1 -4683.075,E2 -4683.075} C_VEL
LIN {X 0,Y 524.037,Z 442.455,A -85,B 0,C 180,E1 -4686.159,E2 -4686.159} C_VEL
LIN {X 0,Y 523.995,Z 442.456,A -85,B 0,C 180,E1 -4689.262,E2 -4689.262} C_VEL
LIN {X 0,Y 523.999,Z 442.464,A -85,B 0,C 180,E1 -4691.743,E2 -4691.743} C_VEL
LIN {X 0,Y 523.983,Z 442.46,A -85,B 0,C 180,E1 -4695.053,E2 -4695.053} C_VEL
LIN {X 0,Y 523.955,Z 442.459,A -85,B 0,C 180,E1 -4697.969,E2 -4697.969} C_VEL
LIN {X 0,Y 523.964,Z 442.449,A -85,B 0,C 180,E1 -4700.41,E2 -4700.41} C_VEL
LIN {X 0,Y 523.908,Z 442.467,A -85,B 0,C 180,E1 -4702.894,E2 -4702.894} C_VEL
LIN {X 0,Y 523.946,Z 442.467,A -85,B 0,C 180,E1 -4705.419,E2 -4705.419} C_VEL
LIN {X 0,Y 523.963,Z 442.453,A -85,B 0,C 180,E1 -4707.999,E2 -4707.999} C_VEL
LIN {X 0,Y 523.945,Z 442.465,A -85,B 0,C 180,E1 -4710.857,E2 -4710.857} C_VEL
LIN {X 0,Y 523.954,Z 442.467,A -85,B 0,C 180,E1 -4713.735,E2 -4713.735} C_VEL
LIN {X 0,Y 523.918,Z 442.474,A -85,B 0,C 180,E1 -4716.405,E2 -4716.405} C_VEL
LIN {X 0,Y 523.925,Z 442.464,A -85,B 0,C 180,E1 -4719.084,E2 -4719.084} C_VEL
LIN {X 0,Y 523.951,Z 442.472,A -85,B 0,C 180,E1 -4722.119,E2 -4722.119} C_VEL
LIN {X 0,Y 523.949,Z 442.465,A -85,B 0,C 180,E1 -4725.309,E2 -4725.309} C_VEL
LIN {X 0,Y 523.956,Z 442.471,A -85,B 0,C 180,E1 -4728.69,E2 -4728.69} C_VEL
LIN {X 0,Y 523.911,Z 442.452,A -85,B 0,C 180,E1 -4731.899,E2 -4731.899} C_VEL
LIN {X 0,Y 523.935,Z 442.465,A -85,B 0,C 180,E1 -4734.909,E2 -4734.909} C_VEL
LIN {X 0,Y 523.981,Z 442.652,A -85,B 0,C 180,E1 -4736.766,E2 -4736.766} C_VEL
LIN {X 0,Y 527.665,Z 456.917,A -85,B 0,C 180,E1 -4739.151,E2 -4739.151} C_VEL
LIN {X 0,Y 528.056,Z 459.983,A -85,B 0,C 180,E1 -4739.62,E2 -4739.62} C_VEL
LIN {X 0,Y 527.316,Z 479.731,A -85,B 0,C 180,E1 -4742.411,E2 -4742.411} C_VEL
LIN {X 0,Y 527.249,Z 484.413,A -85,B 0,C 180,E1 -4743.038,E2 -4743.038} C_VEL
LIN {X 0,Y 531.513,Z 501.706,A -85,B 0,C 180,E1 -4743.543,E2 -4743.543} C_VEL
LIN {X 0,Y 529.957,Z 689.851,A -85,B 0,C 180,E1 -4746.223,E2 -4746.223} C_VEL
LIN {X 0,Y 529.649,Z 705.56,A -85,B 0,C 180,E1 -4746.524,E2 -4746.524} C_VEL
LIN {X 0,Y 529.309,Z 719.737,A -85,B 0,C 180,E1 -4746.915,E2 -4746.915} C_VEL
LIN {X 0,Y 528.887,Z 733.064,A -85,B 0,C 180,E1 -4747.386,E2 -4747.386} C_VEL
LIN {X 0,Y 528.398,Z 746.645,A -85,B 0,C 180,E1 -4747.982,E2 -4747.982} C_VEL
LIN {X 0,Y 527.883,Z 759.309,A -85,B 0,C 180,E1 -4748.65,E2 -4748.65} C_VEL
LIN {X 0,Y 527.345,Z 771.777,A -85,B 0,C 180,E1 -4749.421,E2 -4749.421} C_VEL
LIN {X 0,Y 526.798,Z 782.852,A -85,B 0,C 180,E1 -4750.213,E2 -4750.213} C_VEL
LIN {X 0,Y 526.232,Z 794.908,A -85,B 0,C 180,E1 -4751.205,E2 -4751.205} C_VEL
LIN {X 0,Y 525.628,Z 806.418,A -85,B 0,C 180,E1 -4752.291,E2 -4752.291} C_VEL
LIN {X 0,Y 525.058,Z 819.014,A -85,B 0,C 180,E1 -4753.675,E2 -4753.675} C_VEL
LIN {X 0,Y 524.639,Z 829.5,A -85,B 0,C 180,E1 -4755.03,E2 -4755.03} C_VEL
LIN {X 0,Y 524.229,Z 838.89,A -85,B 0,C 180,E1 -4756.432,E2 -4756.432} C_VEL
LIN {X 0,Y 523.949,Z 846.827,A -85,B 0,C 180,E1 -4757.804,E2 -4757.804} C_VEL
LIN {X 0,Y 523.732,Z 853.647,A -85,B 0,C 180,E1 -4759.172,E2 -4759.172} C_VEL
LIN {X 0,Y 523.544,Z 860.254,A -85,B 0,C 180,E1 -4760.73,E2 -4760.73} C_VEL
LIN {X 0,Y 523.468,Z 865.666,A -85,B 0,C 180,E1 -4762.284,E2 -4762.284} C_VEL
LIN {X 0,Y 523.411,Z 870.011,A -85,B 0,C 180,E1 -4763.834,E2 -4763.834} C_VEL
LIN {X 0,Y 523.31,Z 873.307,A -85,B 0,C 180,E1 -4765.378,E2 -4765.378} C_VEL
LIN {X 0,Y 523.355,Z 875.653,A -85,B 0,C 180,E1 -4766.921,E2 -4766.921} C_VEL
LIN {X 0,Y 523.268,Z 877.021,A -85,B 0,C 180,E1 -4768.461,E2 -4768.461} C_VEL
LIN {X 0,Y 523.241,Z 877.5,A -85,B 0,C 180,E1 -4770,E2 -4770} C_VEL
LIN {X 0,Y 523.268,Z 877.021,A -85,B 0,C 180,E1 -4771.539,E2 -4771.539} C_VEL
LIN {X 0,Y 523.355,Z 875.653,A -85,B 0,C 180,E1 -4773.079,E2 -4773.079} C_VEL
LIN {X 0,Y 523.309,Z 873.307,A -85,B 0,C 180,E1 -4774.622,E2 -4774.622} C_VEL
LIN {X 0,Y 523.449,Z 869.091,A -85,B 0,C 180,E1 -4776.514,E2 -4776.514} C_VEL
LIN {X 0,Y 523.468,Z 865.666,A -85,B 0,C 180,E1 -4777.716,E2 -4777.716} C_VEL
LIN {X 0,Y 523.544,Z 860.254,A -85,B 0,C 180,E1 -4779.27,E2 -4779.27} C_VEL
LIN {X 0,Y 523.732,Z 853.647,A -85,B 0,C 180,E1 -4780.828,E2 -4780.828} C_VEL
LIN {X 0,Y 523.988,Z 845.783,A -85,B 0,C 180,E1 -4782.392,E2 -4782.392} C_VEL
LIN {X 0,Y 524.313,Z 836.448,A -85,B 0,C 180,E1 -4783.962,E2 -4783.962} C_VEL
LIN {X 0,Y 524.828,Z 825.291,A -85,B 0,C 180,E1 -4785.534,E2 -4785.534} C_VEL
LIN {X 0,Y 525.212,Z 815.562,A -85,B 0,C 180,E1 -4786.72,E2 -4786.72} C_VEL
LIN {X 0,Y 525.731,Z 804.416,A -85,B 0,C 180,E1 -4787.906,E2 -4787.906} C_VEL
LIN {X 0,Y 526.324,Z 792.632,A -85,B 0,C 180,E1 -4788.994,E2 -4788.994} C_VEL
LIN {X 0,Y 526.905,Z 780.253,A -85,B 0,C 180,E1 -4789.986,E2 -4789.986} C_VEL
LIN {X 0,Y 527.651,Z 764.119,A -85,B 0,C 180,E1 -4791.077,E2 -4791.077} C_VEL
LIN {X 0,Y 528.296,Z 748.692,A -85,B 0,C 180,E1 -4791.92,E2 -4791.92} C_VEL
LIN {X 0,Y 528.832,Z 735.527,A -85,B 0,C 180,E1 -4792.513,E2 -4792.513} C_VEL
LIN {X 0,Y 529.214,Z 722.797,A -85,B 0,C 180,E1 -4792.986,E2 -4792.986} C_VEL
LIN {X 0,Y 529.569,Z 709.26,A -85,B 0,C 180,E1 -4793.383,E2 -4793.383} C_VEL
LIN {X 0,Y 529.854,Z 696.064,A -85,B 0,C 180,E1 -4793.669,E2 -4793.669} C_VEL
LIN {X 0,Y 530.578,Z 614.798,A -85,B 0,C 180,E1 -4794.843,E2 -4794.843} C_VEL
LIN {X 0,Y 531.364,Z 500.81,A -85,B 0,C 180,E1 -4796.478,E2 -4796.478} C_VEL
LIN {X 0,Y 527.213,Z 484.195,A -85,B 0,C 180,E1 -4796.978,E2 -4796.978} C_VEL
LIN {X 0,Y 527.981,Z 462.925,A -85,B 0,C 180,E1 -4799.96,E2 -4799.96} C_VEL
LIN {X 0,Y 527.979,Z 458.454,A -85,B 0,C 180,E1 -4800.606,E2 -4800.606} C_VEL
LIN {X 0,Y 524.482,Z 444.606,A -85,B 0,C 180,E1 -4802.866,E2 -4802.866} C_VEL
LIN {X 0,Y 523.984,Z 442.568,A -85,B 0,C 180,E1 -4803.245,E2 -4803.245} C_VEL
LIN {X 0,Y 523.918,Z 442.471,A -85,B 0,C 180,E1 -4806.404,E2 -4806.404} C_VEL
LIN {X 0,Y 523.918,Z 442.459,A -85,B 0,C 180,E1 -4809.084,E2 -4809.084} C_VEL
LIN {X 0,Y 523.948,Z 442.465,A -85,B 0,C 180,E1 -4812.118,E2 -4812.118} C_VEL
LIN {X 0,Y 523.95,Z 442.468,A -85,B 0,C 180,E1 -4815.308,E2 -4815.308} C_VEL
LIN {X 0,Y 523.966,Z 442.462,A -85,B 0,C 180,E1 -4818.687,E2 -4818.687} C_VEL
LIN {X 0,Y 523.919,Z 442.466,A -85,B 0,C 180,E1 -4821.079,E2 -4821.079} C_VEL
LIN {X 0,Y 523.923,Z 442.469,A -85,B 0,C 180,E1 -4823.827,E2 -4823.827} C_VEL
LIN {X 0,Y 523.935,Z 442.466,A -85,B 0,C 180,E1 -4826.635,E2 -4826.635} C_VEL
LIN {X 0,Y 523.956,Z 442.464,A -85,B 0,C 180,E1 -4829.356,E2 -4829.356} C_VEL
LIN {X 0,Y 523.972,Z 442.454,A -85,B 0,C 180,E1 -4832.28,E2 -4832.28} C_VEL
LIN {X 0,Y 523.946,Z 442.467,A -85,B 0,C 180,E1 -4834.581,E2 -4834.581} C_VEL
LIN {X 0,Y 523.908,Z 442.467,A -85,B 0,C 180,E1 -4837.106,E2 -4837.106} C_VEL
LIN {X 0,Y 523.97,Z 442.448,A -85,B 0,C 180,E1 -4839.865,E2 -4839.865} C_VEL
LIN {X 0,Y 523.961,Z 442.462,A -85,B 0,C 180,E1 -4842.837,E2 -4842.837} C_VEL
LIN {X 0,Y 523.967,Z 442.461,A -85,B 0,C 180,E1 -4845.235,E2 -4845.235} C_VEL
LIN {X 0,Y 524.002,Z 442.466,A -85,B 0,C 180,E1 -4848.394,E2 -4848.394} C_VEL
LIN {X 0,Y 523.998,Z 442.453,A -85,B 0,C 180,E1 -4851.516,E2 -4851.516} C_VEL
LIN {X 0,Y 524.076,Z 442.453,A -85,B 0,C 180,E1 -4854.613,E2 -4854.613} C_VEL
LIN {X 0,Y 524.103,Z 442.444,A -85,B 0,C 180,E1 -4857.694,E2 -4857.694} C_VEL
LIN {X 0,Y 524.116,Z 442.442,A -85,B 0,C 180,E1 -4860.768,E2 -4860.768} C_VEL
LIN {X 0,Y 524.067,Z 442.451,A -85,B 0,C 180,E1 -4863.075,E2 -4863.075} C_VEL
LIN {X 0,Y 524.042,Z 442.452,A -85,B 0,C 180,E1 -4866.159,E2 -4866.159} C_VEL
LIN {X 0,Y 523.994,Z 442.458,A -85,B 0,C 180,E1 -4869.262,E2 -4869.262} C_VEL
LIN {X 0,Y 523.998,Z 442.454,A -85,B 0,C 180,E1 -4871.743,E2 -4871.743} C_VEL
LIN {X 0,Y 523.983,Z 442.459,A -85,B 0,C 180,E1 -4875.053,E2 -4875.053} C_VEL
LIN {X 0,Y 523.955,Z 442.464,A -85,B 0,C 180,E1 -4877.969,E2 -4877.969} C_VEL
LIN {X 0,Y 523.963,Z 442.464,A -85,B 0,C 180,E1 -4880.41,E2 -4880.41} C_VEL
LIN {X 0,Y 523.907,Z 442.478,A -85,B 0,C 180,E1 -4882.893,E2 -4882.893} C_VEL
LIN {X 0,Y 523.945,Z 442.454,A -85,B 0,C 180,E1 -4885.419,E2 -4885.419} C_VEL
LIN {X 0,Y 523.961,Z 442.455,A -85,B 0,C 180,E1 -4887.999,E2 -4887.999} C_VEL
LIN {X 0,Y 523.943,Z 442.473,A -85,B 0,C 180,E1 -4890.857,E2 -4890.857} C_VEL
LIN {X 0,Y 523.952,Z 442.449,A -85,B 0,C 180,E1 -4893.735,E2 -4893.735} C_VEL
LIN {X 0,Y 523.914,Z 442.468,A -85,B 0,C 180,E1 -4896.405,E2 -4896.405} C_VEL
LIN {X 0,Y 523.952,Z 442.473,A -85,B 0,C 180,E1 -4899.081,E2 -4899.081} C_VEL
LIN {X 0,Y 523.957,Z 442.465,A -85,B 0,C 180,E1 -4902.118,E2 -4902.118} C_VEL
LIN {X 0,Y 523.948,Z 442.473,A -85,B 0,C 180,E1 -4905.309,E2 -4905.309} C_VEL
LIN {X 0,Y 523.911,Z 442.473,A -85,B 0,C 180,E1 -4906.923,E2 -4906.923} C_VEL
LIN {X 0,Y 523.25,Z 442.558,A -85,B 0,C 180,E1 -4907.564,E2 -4907.564} C_VEL
LIN {X 0,Y 520.422,Z 442.907,A -85,B 0,C 180,E1 -4908.606,E2 -4908.606} C_VEL
LIN {X 0,Y 518.024,Z 443.21,A -85,B 0,C 180,E1 -4909.446,E2 -4909.446} C_VEL
LIN {X 0,Y 516.984,Z 443.334,A -85,B 0,C 180,E1 -4910.093,E2 -4910.093} C_VEL
LIN {X 0,Y 516.894,Z 443.344,A -85,B 0,C 180,E1 -4910.313,E2 -4910.313} C_VEL
LIN {X 0,Y 516.878,Z 443.353,A -85,B 0,C 180,E1 -4913.342,E2 -4913.342} C_VEL
LIN {X 0,Y 516.908,Z 443.344,A -85,B 0,C 180,E1 -4916.122,E2 -4916.122} C_VEL
LIN {X 0,Y 516.887,Z 443.348,A -85,B 0,C 180,E1 -4918.936,E2 -4918.936} C_VEL
LIN {X 0,Y 516.915,Z 443.349,A -85,B 0,C 180,E1 -4921.585,E2 -4921.585} C_VEL
LIN {X 0,Y 516.928,Z 443.342,A -85,B 0,C 180,E1 -4924.211,E2 -4924.211} C_VEL
LIN {X 0,Y 516.867,Z 443.349,A -85,B 0,C 180,E1 -4926.777,E2 -4926.777} C_VEL
LIN {X 0,Y 516.935,Z 443.346,A -85,B 0,C 180,E1 -4929.732,E2 -4929.732} C_VEL
LIN {X 0,Y 516.925,Z 443.341,A -85,B 0,C 180,E1 -4932.596,E2 -4932.596} C_VEL
LIN {X 0,Y 516.938,Z 443.341,A -85,B 0,C 180,E1 -4935.03,E2 -4935.03} C_VEL
LIN {X 0,Y 517.001,Z 443.336,A -85,B 0,C 180,E1 -4938.235,E2 -4938.235} C_VEL
LIN {X 0,Y 516.965,Z 443.339,A -85,B 0,C 180,E1 -4941.4,E2 -4941.4} C_VEL
LIN {X 0,Y 517.006,Z 443.337,A -85,B 0,C 180,E1 -4943.757,E2 -4943.757} C_VEL
LIN {X 0,Y 517.081,Z 443.327,A -85,B 0,C 180,E1 -4947.663,E2 -4947.663} C_VEL
LIN {X 0,Y 517.089,Z 443.322,A -85,B 0,C 180,E1 -4950.779,E2 -4950.779} C_VEL
LIN {X 0,Y 517.011,Z 443.331,A -85,B 0,C 180,E1 -4953.117,E2 -4953.117} C_VEL
LIN {X 0,Y 517.006,Z 443.337,A -85,B 0,C 180,E1 -4956.243,E2 -4956.243} C_VEL
LIN {X 0,Y 516.949,Z 443.339,A -85,B 0,C 180,E1 -4959.389,E2 -4959.389} C_VEL
LIN {X 0,Y 516.98,Z 443.339,A -85,B 0,C 180,E1 -4961.824,E2 -4961.824} C_VEL
LIN {X 0,Y 516.94,Z 443.34,A -85,B 0,C 180,E1 -4965.146,E2 -4965.146} C_VEL
LIN {X 0,Y 516.922,Z 443.348,A -85,B 0,C 180,E1 -4968.222,E2 -4968.222} C_VEL
LIN {X 0,Y 516.908,Z 443.347,A -85,B 0,C 180,E1 -4970.701,E2 -4970.701} C_VEL
LIN {X 0,Y 516.898,Z 443.35,A -85,B 0,C 180,E1 -4974.072,E2 -4974.072} C_VEL
LIN {X 0,Y 516.924,Z 443.346,A -85,B 0,C 180,E1 -4976.657,E2 -4976.657} C_VEL
LIN {X 0,Y 516.906,Z 443.344,A -85,B 0,C 180,E1 -4979.524,E2 -4979.524} C_VEL
LIN {X 0,Y 516.895,Z 443.351,A -85,B 0,C 180,E1 -4982.544,E2 -4982.544} C_VEL
LIN {X 0,Y 516.877,Z 443.347,A -85,B 0,C 180,E1 -4985.332,E2 -4985.332} C_VEL
LIN {X 0,Y 516.874,Z 443.348,A -85,B 0,C 180,E1 -4987.943,E2 -4987.943} C_VEL
LIN {X 0,Y 516.897,Z 443.352,A -85,B 0,C 180,E1 -4990.739,E2 -4990.739} C_VEL
LIN {X 0,Y 516.875,Z 443.347,A -85,B 0,C 180,E1 -4993.903,E2 -4993.903} C_VEL
LIN {X 0,Y 516.874,Z 443.348,A -85,B 0,C 180,E1 -4996.107,E2 -4996.107} C_VEL
LIN {X 0,Y 516.9,Z 443.347,A -85,B 0,C 180,E1 -4999.26,E2 -4999.26} C_VEL
LIN {X 0,Y 516.876,Z 443.347,A -85,B 0,C 180,E1 -5002.056,E2 -5002.056} C_VEL
LIN {X 0,Y 516.886,Z 443.333,A -85,B 0,C 180,E1 -5005.176,E2 -5005.176} C_VEL
LIN {X 0,Y 516.873,Z 443.343,A -85,B 0,C 180,E1 -5007.976,E2 -5007.976} C_VEL
LIN {X 0,Y 516.927,Z 443.344,A -85,B 0,C 180,E1 -5010.696,E2 -5010.696} C_VEL
LIN {X 0,Y 516.935,Z 443.325,A -85,B 0,C 180,E1 -5013.803,E2 -5013.803} C_VEL
LIN {X 0,Y 516.862,Z 443.35,A -85,B 0,C 180,E1 -5016.776,E2 -5016.776} C_VEL
LIN {X 0,Y 516.929,Z 443.338,A -85,B 0,C 180,E1 -5019.731,E2 -5019.731} C_VEL
LIN {X 0,Y 516.921,Z 443.342,A -85,B 0,C 180,E1 -5022.596,E2 -5022.596} C_VEL
LIN {X 0,Y 516.94,Z 443.338,A -85,B 0,C 180,E1 -5025.03,E2 -5025.03} C_VEL
LIN {X 0,Y 516.955,Z 443.331,A -85,B 0,C 180,E1 -5028.234,E2 -5028.234} C_VEL
LIN {X 0,Y 516.963,Z 443.342,A -85,B 0,C 180,E1 -5031.4,E2 -5031.4} C_VEL
LIN {X 0,Y 517.038,Z 443.322,A -85,B 0,C 180,E1 -5034.54,E2 -5034.54} C_VEL
LIN {X 0,Y 517.075,Z 443.321,A -85,B 0,C 180,E1 -5037.663,E2 -5037.663} C_VEL
LIN {X 0,Y 517.086,Z 443.32,A -85,B 0,C 180,E1 -5040.779,E2 -5040.779} C_VEL
LIN {X 0,Y 517.008,Z 443.33,A -85,B 0,C 180,E1 -5043.117,E2 -5043.117} C_VEL
LIN {X 0,Y 517,Z 443.331,A -85,B 0,C 180,E1 -5046.243,E2 -5046.243} C_VEL
LIN {X 0,Y 516.949,Z 443.335,A -85,B 0,C 180,E1 -5049.389,E2 -5049.389} C_VEL
LIN {X 0,Y 516.947,Z 443.341,A -85,B 0,C 180,E1 -5051.81,E2 -5051.81} C_VEL
LIN {X 0,Y 516.934,Z 443.339,A -85,B 0,C 180,E1 -5055.147,E2 -5055.147} C_VEL
LIN {X 0,Y 516.917,Z 443.331,A -85,B 0,C 180,E1 -5058.223,E2 -5058.223} C_VEL
LIN {X 0,Y 516.904,Z 443.326,A -85,B 0,C 180,E1 -5060.702,E2 -5060.702} C_VEL
LIN {X 0,Y 516.903,Z 443.35,A -85,B 0,C 180,E1 -5064.072,E2 -5064.072} C_VEL
LIN {X 0,Y 516.921,Z 443.332,A -85,B 0,C 180,E1 -5066.658,E2 -5066.658} C_VEL
LIN {X 0,Y 516.912,Z 443.331,A -85,B 0,C 180,E1 -5069.526,E2 -5069.526} C_VEL
LIN {X 0,Y 516.893,Z 443.345,A -85,B 0,C 180,E1 -5072.545,E2 -5072.545} C_VEL
LIN {X 0,Y 516.875,Z 443.336,A -85,B 0,C 180,E1 -5075.333,E2 -5075.333} C_VEL
LIN {X 0,Y 516.876,Z 443.353,A -85,B 0,C 180,E1 -5077.944,E2 -5077.944} C_VEL
LIN {X 0,Y 516.898,Z 443.344,A -85,B 0,C 180,E1 -5080.74,E2 -5080.74} C_VEL
LIN {X 0,Y 516.877,Z 443.347,A -85,B 0,C 180,E1 -5083.904,E2 -5083.904} C_VEL
LIN {X 0,Y 516.876,Z 443.353,A -85,B 0,C 180,E1 -5086.108,E2 -5086.108} C_VEL
LIN {X 0,Y 516.912,Z 443.345,A -85,B 0,C 180,E1 -5088.399,E2 -5088.399} C_VEL
LIN {X 0,Y 516.877,Z 443.332,A -85,B 0,C 180,E1 -5091.285,E2 -5091.285} C_VEL
LIN {X 0,Y 516.887,Z 443.353,A -85,B 0,C 180,E1 -5094.222,E2 -5094.222} C_VEL
LIN {X 0,Y 516.94,Z 443.501,A -85,B 0,C 180,E1 -5096.417,E2 -5096.417} C_VEL
LIN {X 0,Y 518.735,Z 450.625,A -85,B 0,C 180,E1 -5097.666,E2 -5097.666} C_VEL
LIN {X 0,Y 521.291,Z 460.884,A -85,B 0,C 180,E1 -5099.349,E2 -5099.349} C_VEL
LIN {X 0,Y 520.533,Z 481.076,A -85,B 0,C 180,E1 -5102.238,E2 -5102.238} C_VEL
LIN {X 0,Y 520.457,Z 484.297,A -85,B 0,C 180,E1 -5102.657,E2 -5102.657} C_VEL
LIN {X 0,Y 525.086,Z 502.514,A -85,B 0,C 180,E1 -5103.206,E2 -5103.206} C_VEL
LIN {X 0,Y 523.774,Z 654.149,A -85,B 0,C 180,E1 -5105.395,E2 -5105.395} C_VEL
LIN {X 0,Y 523.336,Z 696.213,A -85,B 0,C 180,E1 -5106.021,E2 -5106.021} C_VEL
LIN {X 0,Y 523.018,Z 710.231,A -85,B 0,C 180,E1 -5106.332,E2 -5106.332} C_VEL
LIN {X 0,Y 522.555,Z 726.605,A -85,B 0,C 180,E1 -5106.835,E2 -5106.835} C_VEL
LIN {X 0,Y 521.908,Z 743.563,A -85,B 0,C 180,E1 -5107.537,E2 -5107.537} C_VEL
LIN {X 0,Y 521.384,Z 755.954,A -85,B 0,C 180,E1 -5108.17,E2 -5108.17} C_VEL
LIN {X 0,Y 520.792,Z 769.082,A -85,B 0,C 180,E1 -5108.964,E2 -5108.964} C_VEL
LIN {X 0,Y 520.122,Z 781.545,A -85,B 0,C 180,E1 -5109.845,E2 -5109.845} C_VEL
LIN {X 0,Y 519.516,Z 792.625,A -85,B 0,C 180,E1 -5110.747,E2 -5110.747} C_VEL
LIN {X 0,Y 519.008,Z 802.856,A -85,B 0,C 180,E1 -5111.696,E2 -5111.696} C_VEL
LIN {X 0,Y 518.404,Z 813.793,A -85,B 0,C 180,E1 -5112.851,E2 -5112.851} C_VEL
LIN {X 0,Y 517.929,Z 823.729,A -85,B 0,C 180,E1 -5114.051,E2 -5114.051} C_VEL
LIN {X 0,Y 517.599,Z 832.418,A -85,B 0,C 180,E1 -5115.251,E2 -5115.251} C_VEL
LIN {X 0,Y 517.186,Z 840.083,A -85,B 0,C 180,E1 -5116.444,E2 -5116.444} C_VEL
LIN {X 0,Y 516.896,Z 847.863,A -85,B 0,C 180,E1 -5117.834,E2 -5117.834} C_VEL
LIN {X 0,Y 516.643,Z 855.439,A -85,B 0,C 180,E1 -5119.418,E2 -5119.418} C_VEL
LIN {X 0,Y 516.449,Z 863.128,A -85,B 0,C 180,E1 -5121.391,E2 -5121.391} C_VEL
LIN {X 0,Y 516.385,Z 867.96,A -85,B 0,C 180,E1 -5122.964,E2 -5122.964} C_VEL
LIN {X 0,Y 516.303,Z 871.755,A -85,B 0,C 180,E1 -5124.532,E2 -5124.532} C_VEL
LIN {X 0,Y 516.302,Z 874.542,A -85,B 0,C 180,E1 -5126.097,E2 -5126.097} C_VEL
LIN {X 0,Y 516.254,Z 876.403,A -85,B 0,C 180,E1 -5127.659,E2 -5127.659} C_VEL
LIN {X 0,Y 516.155,Z 877.318,A -85,B 0,C 180,E1 -5129.22,E2 -5129.22} C_VEL
LIN {X 0,Y 516.155,Z 877.318,A -85,B 0,C 180,E1 -5130.78,E2 -5130.78} C_VEL
LIN {X 0,Y 516.254,Z 876.403,A -85,B 0,C 180,E1 -5132.341,E2 -5132.341} C_VEL
LIN {X 0,Y 516.302,Z 874.542,A -85,B 0,C 180,E1 -5133.903,E2 -5133.903} C_VEL
LIN {X 0,Y 516.303,Z 871.755,A -85,B 0,C 180,E1 -5135.468,E2 -5135.468} C_VEL
LIN {X 0,Y 516.388,Z 866.896,A -85,B 0,C 180,E1 -5137.429,E2 -5137.429} C_VEL
LIN {X 0,Y 516.454,Z 861.75,A -85,B 0,C 180,E1 -5139.003,E2 -5139.003} C_VEL
LIN {X 0,Y 516.643,Z 855.439,A -85,B 0,C 180,E1 -5140.582,E2 -5140.582} C_VEL
LIN {X 0,Y 516.895,Z 847.863,A -85,B 0,C 180,E1 -5142.166,E2 -5142.166} C_VEL
LIN {X 0,Y 517.186,Z 840.083,A -85,B 0,C 180,E1 -5143.556,E2 -5143.556} C_VEL
LIN {X 0,Y 517.613,Z 831.05,A -85,B 0,C 180,E1 -5144.95,E2 -5144.95} C_VEL
LIN {X 0,Y 518.074,Z 820.62,A -85,B 0,C 180,E1 -5146.349,E2 -5146.349} C_VEL
LIN {X 0,Y 518.687,Z 808.387,A -85,B 0,C 180,E1 -5147.75,E2 -5147.75} C_VEL
LIN {X 0,Y 519.353,Z 796.039,A -85,B 0,C 180,E1 -5148.951,E2 -5148.951} C_VEL
LIN {X 0,Y 519.982,Z 784.144,A -85,B 0,C 180,E1 -5149.954,E2 -5149.954} C_VEL
LIN {X 0,Y 520.538,Z 773.404,A -85,B 0,C 180,E1 -5150.747,E2 -5150.747} C_VEL
LIN {X 0,Y 521.155,Z 760.991,A -85,B 0,C 180,E1 -5151.539,E2 -5151.539} C_VEL
LIN {X 0,Y 521.674,Z 748.678,A -85,B 0,C 180,E1 -5152.213,E2 -5152.213} C_VEL
LIN {X 0,Y 522.24,Z 735.512,A -85,B 0,C 180,E1 -5152.813,E2 -5152.813} C_VEL
LIN {X 0,Y 522.683,Z 722.785,A -85,B 0,C 180,E1 -5153.29,E2 -5153.29} C_VEL
LIN {X 0,Y 523.066,Z 709.233,A -85,B 0,C 180,E1 -5153.692,E2 -5153.692} C_VEL
LIN {X 0,Y 523.365,Z 696.276,A -85,B 0,C 180,E1 -5153.976,E2 -5153.976} C_VEL
LIN {X 0,Y 523.932,Z 639.839,A -85,B 0,C 180,E1 -5154.809,E2 -5154.809} C_VEL
LIN {X 0,Y 525.085,Z 502.493,A -85,B 0,C 180,E1 -5156.794,E2 -5156.794} C_VEL
LIN {X 0,Y 520.453,Z 484.076,A -85,B 0,C 180,E1 -5157.357,E2 -5157.357} C_VEL
LIN {X 0,Y 521.263,Z 463.834,A -85,B 0,C 180,E1 -5160.219,E2 -5160.219} C_VEL
LIN {X 0,Y 521.083,Z 459.744,A -85,B 0,C 180,E1 -5160.831,E2 -5160.831} C_VEL
LIN {X 0,Y 516.959,Z 443.536,A -85,B 0,C 180,E1 -5163.553,E2 -5163.553} C_VEL
LIN {X 0,Y 516.878,Z 443.34,A -85,B 0,C 180,E1 -5166.745,E2 -5166.745} C_VEL
LIN {X 0,Y 516.877,Z 443.344,A -85,B 0,C 180,E1 -5169.721,E2 -5169.721} C_VEL
LIN {X 0,Y 516.908,Z 443.344,A -85,B 0,C 180,E1 -5171.774,E2 -5171.774} C_VEL
LIN {X 0,Y 516.917,Z 443.342,A -85,B 0,C 180,E1 -5175.009,E2 -5175.009} C_VEL
LIN {X 0,Y 516.916,Z 443.341,A -85,B 0,C 180,E1 -5178.397,E2 -5178.397} C_VEL
LIN {X 0,Y 516.88,Z 443.344,A -85,B 0,C 180,E1 -5181.284,E2 -5181.284} C_VEL
LIN {X 0,Y 516.884,Z 443.338,A -85,B 0,C 180,E1 -5184.221,E2 -5184.221} C_VEL
LIN {X 0,Y 516.89,Z 443.343,A -85,B 0,C 180,E1 -5187.053,E2 -5187.053} C_VEL
LIN {X 0,Y 516.893,Z 443.344,A -85,B 0,C 180,E1 -5189.796,E2 -5189.796} C_VEL
LIN {X 0,Y 516.922,Z 443.333,A -85,B 0,C 180,E1 -5192.467,E2 -5192.467} C_VEL
LIN {X 0,Y 516.903,Z 443.342,A -85,B 0,C 180,E1 -5195.072,E2 -5195.072} C_VEL
LIN {X 0,Y 516.877,Z 443.334,A -85,B 0,C 180,E1 -5198.462,E2 -5198.462} C_VEL
LIN {X 0,Y 516.896,Z 443.331,A -85,B 0,C 180,E1 -5200.955,E2 -5200.955} C_VEL
LIN {X 0,Y 516.907,Z 443.34,A -85,B 0,C 180,E1 -5203.41,E2 -5203.41} C_VEL
LIN {X 0,Y 516.886,Z 443.346,A -85,B 0,C 180,E1 -5205.833,E2 -5205.833} C_VEL
LIN {X 0,Y 516.948,Z 443.337,A -85,B 0,C 180,E1 -5209.028,E2 -5209.028} C_VEL
LIN {X 0,Y 516.969,Z 443.334,A -85,B 0,C 180,E1 -5212.187,E2 -5212.187} C_VEL
LIN {X 0,Y 517.023,Z 443.332,A -85,B 0,C 180,E1 -5214.54,E2 -5214.54} C_VEL
LIN {X 0,Y 517.075,Z 443.319,A -85,B 0,C 180,E1 -5217.663,E2 -5217.663} C_VEL
LIN {X 0,Y 517.086,Z 443.317,A -85,B 0,C 180,E1 -5220.779,E2 -5220.779} C_VEL
LIN {X 0,Y 517.007,Z 443.33,A -85,B 0,C 180,E1 -5223.117,E2 -5223.117} C_VEL
LIN {X 0,Y 517.005,Z 443.329,A -85,B 0,C 180,E1 -5226.243,E2 -5226.243} C_VEL
LIN {X 0,Y 516.948,Z 443.335,A -85,B 0,C 180,E1 -5229.389,E2 -5229.389} C_VEL
LIN {X 0,Y 516.947,Z 443.332,A -85,B 0,C 180,E1 -5231.81,E2 -5231.81} C_VEL
LIN {X 0,Y 516.936,Z 443.336,A -85,B 0,C 180,E1 -5235.147,E2 -5235.147} C_VEL
LIN {X 0,Y 516.916,Z 443.343,A -85,B 0,C 180,E1 -5238.222,E2 -5238.222} C_VEL
LIN {X 0,Y 516.903,Z 443.345,A -85,B 0,C 180,E1 -5240.702,E2 -5240.702} C_VEL
LIN {X 0,Y 516.901,Z 443.341,A -85,B 0,C 180,E1 -5244.072,E2 -5244.072} C_VEL
LIN {X 0,Y 516.92,Z 443.327,A -85,B 0,C 180,E1 -5246.658,E2 -5246.658} C_VEL
LIN {X 0,Y 516.915,Z 443.343,A -85,B 0,C 180,E1 -5249.527,E2 -5249.527} C_VEL
LIN {X 0,Y 516.891,Z 443.344,A -85,B 0,C 180,E1 -5252.545,E2 -5252.545} C_VEL
LIN {X 0,Y 516.874,Z 443.344,A -85,B 0,C 180,E1 -5255.333,E2 -5255.333} C_VEL
LIN {X 0,Y 516.877,Z 443.347,A -85,B 0,C 180,E1 -5257.944,E2 -5257.944} C_VEL
LIN {X 0,Y 516.9,Z 443.347,A -85,B 0,C 180,E1 -5260.74,E2 -5260.74} C_VEL
LIN {X 0,Y 516.874,Z 443.348,A -85,B 0,C 180,E1 -5263.903,E2 -5263.903} C_VEL
LIN {X 0,Y 516.875,Z 443.347,A -85,B 0,C 180,E1 -5266.107,E2 -5266.107} C_VEL
LIN {X 0,Y 516.897,Z 443.352,A -85,B 0,C 180,E1 -5269.261,E2 -5269.261} C_VEL
LIN {X 0,Y 516.894,Z 443.344,A -85,B 0,C 180,E1 -5270.313,E2 -5270.313} C_VEL
LIN {X 0,Y 516.214,Z 443.434,A -85,B 0,C 180,E1 -5270.963,E2 -5270.963} C_VEL
LIN {X 0,Y 513.36,Z 443.793,A -85,B 0,C 180,E1 -5272.018,E2 -5272.018} C_VEL
LIN {X 0,Y 510.951,Z 444.094,A -85,B 0,C 180,E1 -5272.868,E2 -5272.868} C_VEL
LIN {X 0,Y 509.912,Z 444.221,A -85,B 0,C 180,E1 -5273.525,E2 -5273.525} C_VEL
LIN {X 0,Y 509.825,Z 444.229,A -85,B 0,C 180,E1 -5273.747,E2 -5273.747} C_VEL
LIN {X 0,Y 509.858,Z 444.222,A -85,B 0,C 180,E1 -5276.54,E2 -5276.54} C_VEL
LIN {X 0,Y 509.84,Z 444.229,A -85,B 0,C 180,E1 -5279.335,E2 -5279.335} C_VEL
LIN {X 0,Y 509.89,Z 444.22,A -85,B 0,C 180,E1 -5282.055,E2 -5282.055} C_VEL
LIN {X 0,Y 509.873,Z 444.219,A -85,B 0,C 180,E1 -5284.704,E2 -5284.704} C_VEL
LIN {X 0,Y 509.832,Z 444.23,A -85,B 0,C 180,E1 -5287.455,E2 -5287.455} C_VEL
LIN {X 0,Y 509.912,Z 444.22,A -85,B 0,C 180,E1 -5289.845,E2 -5289.845} C_VEL
LIN {X 0,Y 509.881,Z 444.22,A -85,B 0,C 180,E1 -5293.175,E2 -5293.175} C_VEL
LIN {X 0,Y 509.861,Z 444.227,A -85,B 0,C 180,E1 -5295.634,E2 -5295.634} C_VEL
LIN {X 0,Y 509.918,Z 444.215,A -85,B 0,C 180,E1 -5298.875,E2 -5298.875} C_VEL
LIN {X 0,Y 509.948,Z 444.215,A -85,B 0,C 180,E1 -5302.079,E2 -5302.079} C_VEL
LIN {X 0,Y 509.978,Z 444.209,A -85,B 0,C 180,E1 -5304.464,E2 -5304.464} C_VEL
LIN {X 0,Y 510.052,Z 444.203,A -85,B 0,C 180,E1 -5307.631,E2 -5307.631} C_VEL
LIN {X 0,Y 510.06,Z 444.198,A -85,B 0,C 180,E1 -5310.789,E2 -5310.789} C_VEL
LIN {X 0,Y 509.953,Z 444.211,A -85,B 0,C 180,E1 -5313.16,E2 -5313.16} C_VEL
LIN {X 0,Y 509.975,Z 444.213,A -85,B 0,C 180,E1 -5316.329,E2 -5316.329} C_VEL
LIN {X 0,Y 509.911,Z 444.217,A -85,B 0,C 180,E1 -5318.72,E2 -5318.72} C_VEL
LIN {X 0,Y 509.948,Z 444.215,A -85,B 0,C 180,E1 -5321.93,E2 -5321.93} C_VEL
LIN {X 0,Y 509.89,Z 444.218,A -85,B 0,C 180,E1 -5325.242,E2 -5325.242} C_VEL
LIN {X 0,Y 509.885,Z 444.222,A -85,B 0,C 180,E1 -5328.001,E2 -5328.001} C_VEL
LIN {X 0,Y 509.845,Z 444.224,A -85,B 0,C 180,E1 -5331.001,E2 -5331.001} C_VEL
LIN {X 0,Y 509.86,Z 444.227,A -85,B 0,C 180,E1 -5334.426,E2 -5334.426} C_VEL
LIN {X 0,Y 509.882,Z 444.22,A -85,B 0,C 180,E1 -5337.055,E2 -5337.055} C_VEL
LIN {X 0,Y 509.851,Z 444.223,A -85,B 0,C 180,E1 -5339.751,E2 -5339.751} C_VEL
LIN {X 0,Y 509.871,Z 444.226,A -85,B 0,C 180,E1 -5342.775,E2 -5342.775} C_VEL
LIN {X 0,Y 509.837,Z 444.223,A -85,B 0,C 180,E1 -5345.581,E2 -5345.581} C_VEL
LIN {X 0,Y 509.845,Z 444.228,A -85,B 0,C 180,E1 -5348.337,E2 -5348.337} C_VEL
LIN {X 0,Y 509.858,Z 444.222,A -85,B 0,C 180,E1 -5351.424,E2 -5351.424} C_VEL
LIN {X 0,Y 509.849,Z 444.229,A -85,B 0,C 180,E1 -5354.668,E2 -5354.668} C_VEL
LIN {X 0,Y 509.878,Z 444.219,A -85,B 0,C 180,E1 -5358.099,E2 -5358.099} C_VEL
LIN {X 0,Y 509.868,Z 444.226,A -85,B 0,C 180,E1 -5360.65,E2 -5360.65} C_VEL
LIN {X 0,Y 509.827,Z 444.223,A -85,B 0,C 180,E1 -5363.648,E2 -5363.648} C_VEL
LIN {X 0,Y 509.853,Z 444.205,A -85,B 0,C 180,E1 -5366.539,E2 -5366.539} C_VEL
LIN {X 0,Y 509.842,Z 444.227,A -85,B 0,C 180,E1 -5369.334,E2 -5369.334} C_VEL
LIN {X 0,Y 509.886,Z 444.207,A -85,B 0,C 180,E1 -5372.054,E2 -5372.054} C_VEL
LIN {X 0,Y 509.868,Z 444.207,A -85,B 0,C 180,E1 -5374.704,E2 -5374.704} C_VEL
LIN {X 0,Y 509.846,Z 444.226,A -85,B 0,C 180,E1 -5377.45,E2 -5377.45} C_VEL
LIN {X 0,Y 509.907,Z 444.212,A -85,B 0,C 180,E1 -5379.845,E2 -5379.845} C_VEL
LIN {X 0,Y 509.877,Z 444.221,A -85,B 0,C 180,E1 -5383.175,E2 -5383.175} C_VEL
LIN {X 0,Y 509.863,Z 444.223,A -85,B 0,C 180,E1 -5385.634,E2 -5385.634} C_VEL
LIN {X 0,Y 509.908,Z 444.212,A -85,B 0,C 180,E1 -5388.875,E2 -5388.875} C_VEL
LIN {X 0,Y 509.942,Z 444.208,A -85,B 0,C 180,E1 -5392.079,E2 -5392.079} C_VEL
LIN {X 0,Y 509.987,Z 444.2,A -85,B 0,C 180,E1 -5394.465,E2 -5394.465} C_VEL
LIN {X 0,Y 510.046,Z 444.197,A -85,B 0,C 180,E1 -5397.631,E2 -5397.631} C_VEL
LIN {X 0,Y 510.056,Z 444.196,A -85,B 0,C 180,E1 -5400.79,E2 -5400.79} C_VEL
LIN {X 0,Y 509.95,Z 444.21,A -85,B 0,C 180,E1 -5403.16,E2 -5403.16} C_VEL
LIN {X 0,Y 509.969,Z 444.207,A -85,B 0,C 180,E1 -5406.33,E2 -5406.33} C_VEL
LIN {X 0,Y 509.91,Z 444.206,A -85,B 0,C 180,E1 -5408.72,E2 -5408.72} C_VEL
LIN {X 0,Y 509.896,Z 444.217,A -85,B 0,C 180,E1 -5411.932,E2 -5411.932} C_VEL
LIN {X 0,Y 509.884,Z 444.218,A -85,B 0,C 180,E1 -5415.242,E2 -5415.242} C_VEL
LIN {X 0,Y 509.879,Z 444.21,A -85,B 0,C 180,E1 -5418.001,E2 -5418.001} C_VEL
LIN {X 0,Y 509.842,Z 444.205,A -85,B 0,C 180,E1 -5421.002,E2 -5421.002} C_VEL
LIN {X 0,Y 509.861,Z 444.222,A -85,B 0,C 180,E1 -5424.426,E2 -5424.426} C_VEL
LIN {X 0,Y 509.879,Z 444.208,A -85,B 0,C 180,E1 -5427.056,E2 -5427.056} C_VEL
LIN {X 0,Y 509.872,Z 444.209,A -85,B 0,C 180,E1 -5429.75,E2 -5429.75} C_VEL
LIN {X 0,Y 509.869,Z 444.218,A -85,B 0,C 180,E1 -5432.775,E2 -5432.775} C_VEL
LIN {X 0,Y 509.835,Z 444.214,A -85,B 0,C 180,E1 -5435.582,E2 -5435.582} C_VEL
LIN {X 0,Y 509.846,Z 444.225,A -85,B 0,C 180,E1 -5438.338,E2 -5438.338} C_VEL
LIN {X 0,Y 509.859,Z 444.219,A -85,B 0,C 180,E1 -5441.425,E2 -5441.425} C_VEL
LIN {X 0,Y 509.851,Z 444.222,A -85,B 0,C 180,E1 -5444.668,E2 -5444.668} C_VEL
LIN {X 0,Y 509.853,Z 444.221,A -85,B 0,C 180,E1 -5448.104,E2 -5448.104} C_VEL
LIN {X 0,Y 509.842,Z 444.213,A -85,B 0,C 180,E1 -5450.648,E2 -5450.648} C_VEL
LIN {X 0,Y 509.831,Z 444.225,A -85,B 0,C 180,E1 -5453.648,E2 -5453.648} C_VEL
LIN {X 0,Y 509.894,Z 444.376,A -85,B 0,C 180,E1 -5456.068,E2 -5456.068} C_VEL
LIN {X 0,Y 513.559,Z 458.454,A -85,B 0,C 180,E1 -5458.512,E2 -5458.512} C_VEL
LIN {X 0,Y 514.566,Z 463.758,A -85,B 0,C 180,E1 -5459.368,E2 -5459.368} C_VEL
LIN {X 0,Y 513.689,Z 483.535,A -85,B 0,C 180,E1 -5462.224,E2 -5462.224} C_VEL
LIN {X 0,Y 513.996,Z 485.448,A -85,B 0,C 180,E1 -5462.321,E2 -5462.321} C_VEL
LIN {X 0,Y 518.793,Z 504.325,A -85,B 0,C 180,E1 -5462.884,E2 -5462.884} C_VEL
LIN {X 0,Y 517.065,Z 685.878,A -85,B 0,C 180,E1 -5465.529,E2 -5465.529} C_VEL
LIN {X 0,Y 516.652,Z 704.763,A -85,B 0,C 180,E1 -5465.877,E2 -5465.877} C_VEL
LIN {X 0,Y 516.251,Z 719.714,A -85,B 0,C 180,E1 -5466.296,E2 -5466.296} C_VEL
LIN {X 0,Y 515.777,Z 733.032,A -85,B 0,C 180,E1 -5466.778,E2 -5466.778} C_VEL
LIN {X 0,Y 515.232,Z 745.596,A -85,B 0,C 180,E1 -5467.336,E2 -5467.336} C_VEL
LIN {X 0,Y 514.669,Z 757.856,A -85,B 0,C 180,E1 -5467.986,E2 -5467.986} C_VEL
LIN {X 0,Y 514.083,Z 769.518,A -85,B 0,C 180,E1 -5468.708,E2 -5468.708} C_VEL
LIN {X 0,Y 513.394,Z 781.537,A -85,B 0,C 180,E1 -5469.57,E2 -5469.57} C_VEL
LIN {X 0,Y 512.748,Z 792.618,A -85,B 0,C 180,E1 -5470.483,E2 -5470.483} C_VEL
LIN {X 0,Y 512.169,Z 803.216,A -85,B 0,C 180,E1 -5471.48,E2 -5471.48} C_VEL
LIN {X 0,Y 511.524,Z 813.788,A -85,B 0,C 180,E1 -5472.613,E2 -5472.613} C_VEL
LIN {X 0,Y 510.991,Z 823.723,A -85,B 0,C 180,E1 -5473.829,E2 -5473.829} C_VEL
LIN {X 0,Y 510.621,Z 832.414,A -85,B 0,C 180,E1 -5475.045,E2 -5475.045} C_VEL
LIN {X 0,Y 510.151,Z 841.275,A -85,B 0,C 180,E1 -5476.456,E2 -5476.456} C_VEL
LIN {X 0,Y 509.832,Z 850.396,A -85,B 0,C 180,E1 -5478.16,E2 -5478.16} C_VEL
LIN {X 0,Y 509.475,Z 858.718,A -85,B 0,C 180,E1 -5480.071,E2 -5480.071} C_VEL
LIN {X 0,Y 509.347,Z 864.393,A -85,B 0,C 180,E1 -5481.67,E2 -5481.67} C_VEL
LIN {X 0,Y 509.307,Z 867.956,A -85,B 0,C 180,E1 -5482.866,E2 -5482.866} C_VEL
LIN {X 0,Y 509.214,Z 871.751,A -85,B 0,C 180,E1 -5484.456,E2 -5484.456} C_VEL
LIN {X 0,Y 509.194,Z 874.54,A -85,B 0,C 180,E1 -5486.043,E2 -5486.043} C_VEL
LIN {X 0,Y 509.154,Z 876.399,A -85,B 0,C 180,E1 -5487.627,E2 -5487.627} C_VEL
LIN {X 0,Y 509.068,Z 877.314,A -85,B 0,C 180,E1 -5489.209,E2 -5489.209} C_VEL
LIN {X 0,Y 509.068,Z 877.314,A -85,B 0,C 180,E1 -5490.791,E2 -5490.791} C_VEL
LIN {X 0,Y 509.154,Z 876.399,A -85,B 0,C 180,E1 -5492.373,E2 -5492.373} C_VEL
LIN {X 0,Y 509.194,Z 874.54,A -85,B 0,C 180,E1 -5493.957,E2 -5493.957} C_VEL
